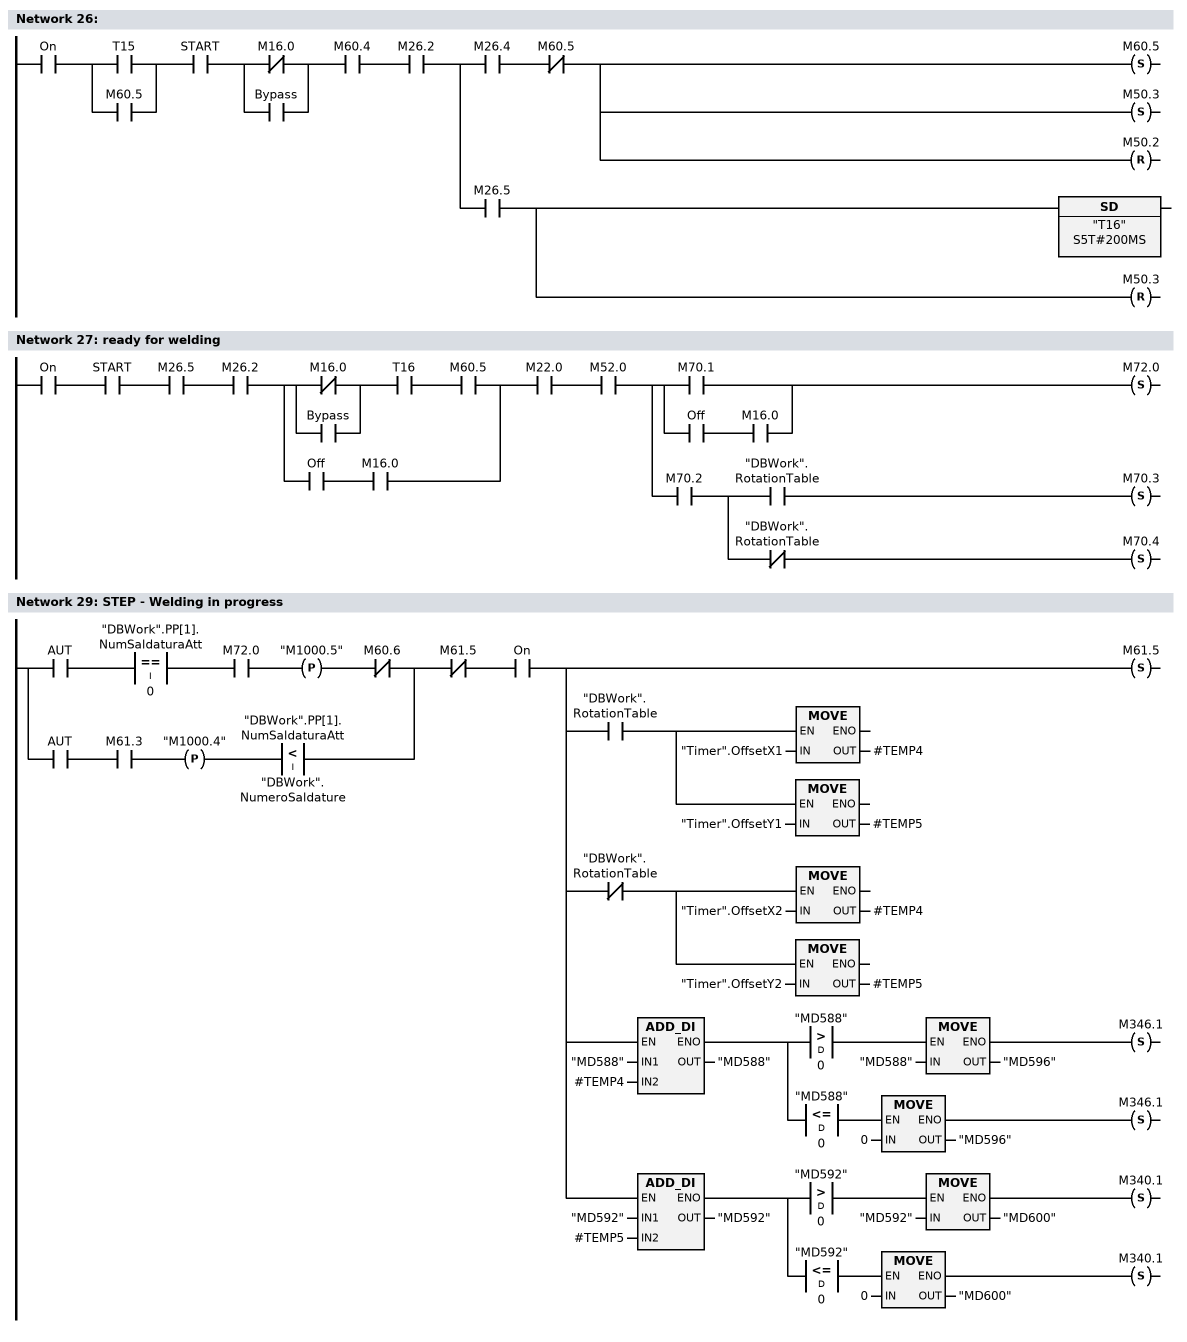
[picture p24: FC14 - AUTOMATIC networks 26-29]
NETWORK
TITLE =
      A     "On";
      A(;
      O     "T15";
      O     "M60.5";
      );
      A     "START";
      A(;
      ON    "M16.0";
      O     "Bypass";
      );
      A     "M60.4";
      A     "M26.2";
      =     L 24.0;
      A     L 24.0;
      A     "M26.4";
      AN    "M60.5";
      S     "M60.5";
      S     "M50.3";
      R     "M50.2";
      A     L 24.0;
      A     "M26.5";
      L     S5T#200MS;
      SD    "T16";
      R     "M50.3";
NETWORK
TITLE = ready for welding
      A     "On";
      A     "START";
      A     "M26.5";
      A     "M26.2";
      A(;
      A(;
      ON    "M16.0";
      O     "Bypass";
      );
      A     "T16";
      A     "M60.5";
      O;
      A     "Off";
      A     "M16.0";
      );
      A     "M22.0";
      A     "M52.0";
      =     L 24.0;
      A     L 24.0;
      A(;
      O     "M70.1";
      O;
      A     "Off";
      A     "M16.0";
      );
      S     "M72.0";
      A     L 24.0;
      A     "M70.2";
      =     L 24.1;
      A     L 24.1;
      A     "DBWork".RotationTable;
      S     "M70.3";
      A     L 24.1;
      AN    "DBWork".RotationTable;
      S     "M70.4";
NETWORK
TITLE =
NETWORK
TITLE = STEP - Welding in progress
      A(;
      A     "AUT";
      A(;
      L     "DBWork".PP[1].NumSaldaturaAtt;
      L     0;
      ==I;
      );
      A     "M72.0";
      FP    "M1000.5";
      AN    "M60.6";
      O(;
      A     "AUT";
      A     "M61.3";
      FP    "M1000.4";
      A(;
      L     "DBWork".PP[1].NumSaldaturaAtt;
      L     "DBWork".NumeroSaldature;
      <I;
      );
      );
      );
      AN    "M61.5";
      A     "On";
      =     L 24.0;
      A     L 24.0;
      BLD   102;
      S     "M61.5";
      A     L 24.0;
      A     "DBWork".RotationTable;
      =     L 24.1;
      A     L 24.1;
      JNB   _00a;
      L     "Timer".OffsetX1;
      T     #TEMP4;
_00a: NOP   0;
      A     L 24.1;
      JNB   _00b;
      L     "Timer".OffsetY1;
      T     #TEMP5;
_00b: NOP   0;
      A     L 24.0;
      AN    "DBWork".RotationTable;
      =     L 24.1;
      A     L 24.1;
      JNB   _00c;
      L     "Timer".OffsetX2;
      T     #TEMP4;
_00c: NOP   0;
      A     L 24.1;
      JNB   _00d;
      L     "Timer".OffsetY2;
      T     #TEMP5;
_00d: NOP   0;
      A     L 24.0;
      JNB   _00e;
      L     "MD588";
      L     #TEMP4;
      +D;
      T     "MD588";
      AN    OV;
      SAVE;
      CLR;
_00e: A     BR;
      =     L 24.1;
      A     L 24.1;
      A(;
      L     "MD588";
      L     0;
      >D;
      );
      JNB   _00f;
      L     "MD588";
      T     "MD596";
      SET;
      SAVE;
      CLR;
_00f: A     BR;
      S     "M346.1";
      A     L 24.1;
      A(;
      L     "MD588";
      L     0;
      <=D;
      );
      JNB   _010;
      L     0;
      T     "MD596";
      SET;
      SAVE;
      CLR;
_010: A     BR;
      S     "M346.1";
      A     L 24.0;
      JNB   _011;
      L     "MD592";
      L     #TEMP5;
      +D;
      T     "MD592";
      AN    OV;
      SAVE;
      CLR;
_011: A     BR;
      =     L 24.1;
      A     L 24.1;
      A(;
      L     "MD592";
      L     0;
      >D;
      );
      JNB   _012;
      L     "MD592";
      T     "MD600";
      SET;
      SAVE;
      CLR;
_012: A     BR;
      S     "M340.1";
      A     L 24.1;
      A(;
      L     "MD592";
      L     0;
      <=D;
      );
      JNB   _013;
      L     0;
      T     "MD600";
      SET;
      SAVE;
      CLR;
_013: A     BR;
      S     "M340.1";
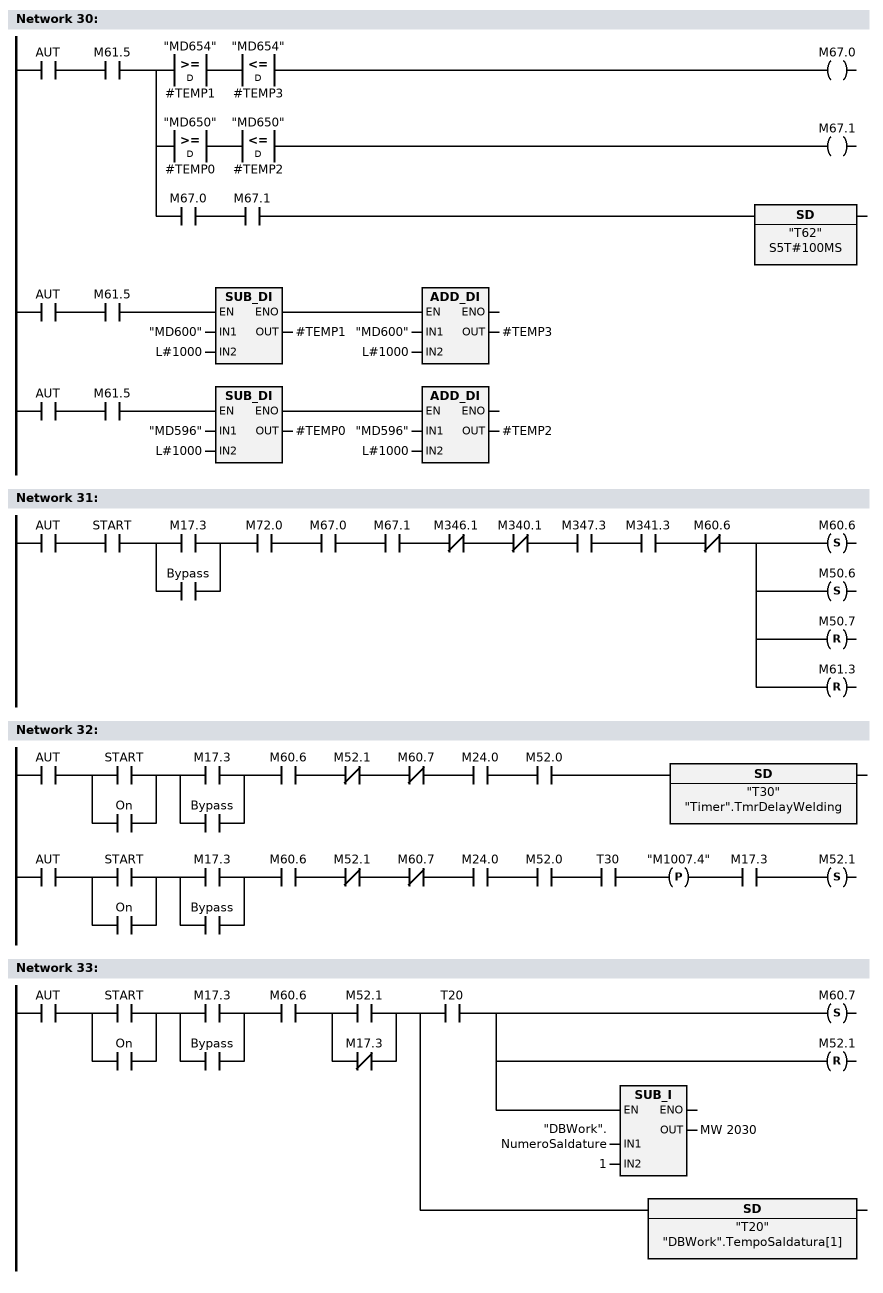
NETWORK
TITLE =
      A     "AUT";
      A     "M61.5";
      =     L 24.0;
      A(;
      A     L 24.0;
      JNB   _014;
      L     "MD600";
      L     L#1000;
      -D;
      T     #TEMP1;
      AN    OV;
      SAVE;
      CLR;
_014: A     BR;
      );
      JNB   _015;
      L     "MD600";
      L     L#1000;
      +D;
      T     #TEMP3;
_015: NOP   0;
      A(;
      A     L 24.0;
      JNB   _016;
      L     "MD596";
      L     L#1000;
      -D;
      T     #TEMP0;
      AN    OV;
      SAVE;
      CLR;
_016: A     BR;
      );
      JNB   _017;
      L     "MD596";
      L     L#1000;
      +D;
      T     #TEMP2;
_017: NOP   0;
      A     L 24.0;
      A(;
      L     "MD654";
      L     #TEMP1;
      >=D;
      );
      A(;
      L     "MD654";
      L     #TEMP3;
      <=D;
      );
      =     "M67.0";
      A     L 24.0;
      A(;
      L     "MD650";
      L     #TEMP0;
      >=D;
      );
      A(;
      L     "MD650";
      L     #TEMP2;
      <=D;
      );
      =     "M67.1";
      A     L 24.0;
      A     "M67.0";
      A     "M67.1";
      L     S5T#100MS;
      SD    "T62";
NETWORK
TITLE =
      A     "AUT";
      A     "START";
      A(;
      O     "M17.3";
      O     "Bypass";
      );
      A     "M72.0";
      A     "M67.0";
      A     "M67.1";
      AN    "M346.1";
      AN    "M340.1";
      A     "M347.3";
      A     "M341.3";
      AN    "M60.6";
      S     "M60.6";
      S     "M50.6";
      R     "M50.7";
      R     "M61.3";
NETWORK
TITLE =
      A     "AUT";
      A(;
      O     "START";
      O     "On";
      );
      A(;
      O     "M17.3";
      O     "Bypass";
      );
      A     "M60.6";
      AN    "M52.1";
      AN    "M60.7";
      A     "M24.0";
      A     "M52.0";
      =     L 24.0;
      A     L 24.0;
      BLD   102;
      L     "Timer".TmrDelayWelding;
      SD    "T30";
      A(;
      A     L 24.0;
      A     "T30";
      FP    "M1007.4";
      );
      A     "M17.3";
      S     "M52.1";
NETWORK
TITLE =
      A     "AUT";
      A(;
      O     "START";
      O     "On";
      );
      A(;
      O     "M17.3";
      O     "Bypass";
      );
      A     "M60.6";
      A(;
      O     "M52.1";
      ON    "M17.3";
      );
      =     L 24.0;
      A     L 24.0;
      A     "T20";
      =     L 24.1;
      A     L 24.1;
      BLD   102;
      S     "M60.7";
      A     L 24.1;
      BLD   102;
      R     "M52.1";
      A     L 24.1;
      JNB   _018;
      L     "DBWork".NumeroSaldature;
      L     1;
      -I;
      T     MW 2030;
_018: NOP   0;
      A     L 24.0;
      BLD   102;
      L     "DBWork".TempoSaldatura[1];
      SD    "T20";
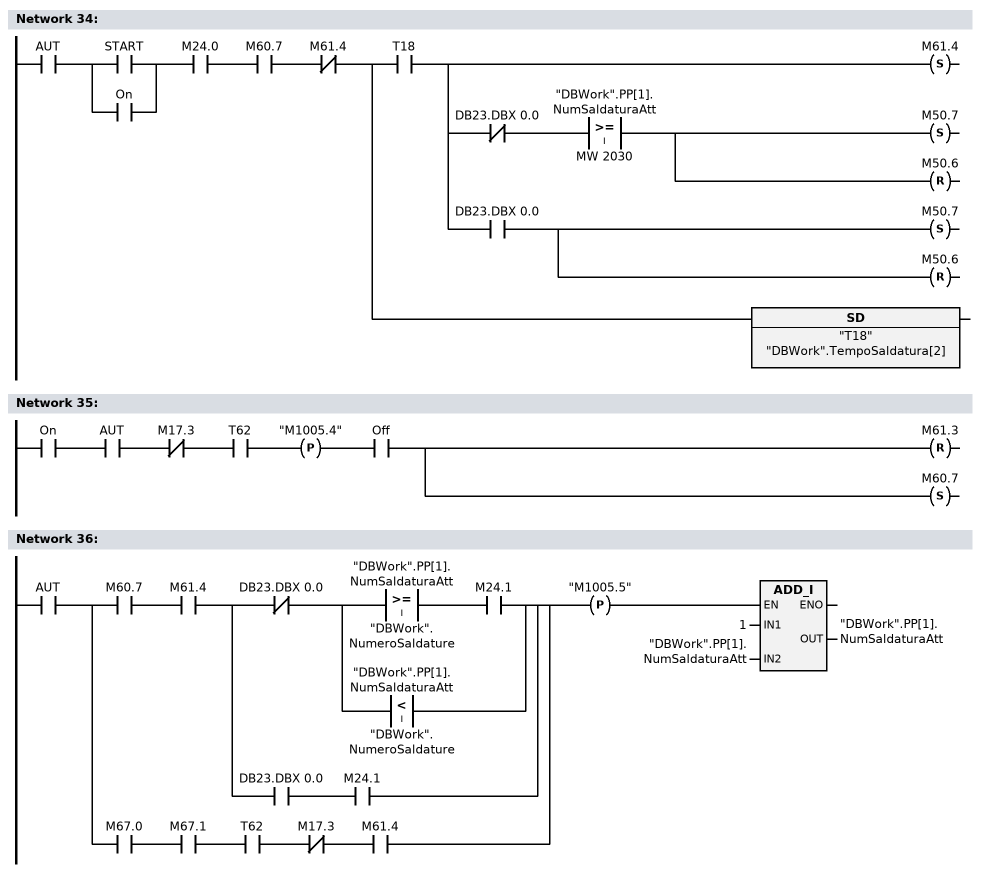
NETWORK
TITLE =
      A     "AUT";
      A(;
      O     "START";
      O     "On";
      );
      A     "M24.0";
      A     "M60.7";
      AN    "M61.4";
      =     L 24.0;
      A     L 24.0;
      A     "T18";
      =     L 24.1;
      A     L 24.1;
      BLD   102;
      S     "M61.4";
      A     L 24.1;
      AN    DB23.DBX 0.0;
      A(;
      L     "DBWork".PP[1].NumSaldaturaAtt;
      L     MW 2030;
      >=I;
      );
      S     "M50.7";
      R     "M50.6";
      A     L 24.1;
      A     DB23.DBX 0.0;
      S     "M50.7";
      R     "M50.6";
      A     L 24.0;
      BLD   102;
      L     "DBWork".TempoSaldatura[2];
      SD    "T18";
NETWORK
TITLE =
      A     "On";
      A     "AUT";
      AN    "M17.3";
      A     "T62";
      FP    "M1005.4";
      A     "Off";
      R     "M61.3";
      S     "M60.7";
NETWORK
TITLE =
      A     "AUT";
      A(;
      A     "M60.7";
      A     "M61.4";
      A(;
      AN    DB23.DBX 0.0;
      A(;
      A(;
      L     "DBWork".PP[1].NumSaldaturaAtt;
      L     "DBWork".NumeroSaldature;
      >=I;
      );
      A     "M24.1";
      O(;
      L     "DBWork".PP[1].NumSaldaturaAtt;
      L     "DBWork".NumeroSaldature;
      <I;
      );
      );
      O;
      A     DB23.DBX 0.0;
      A     "M24.1";
      );
      O;
      A     "M67.0";
      A     "M67.1";
      A     "T62";
      AN    "M17.3";
      A     "M61.4";
      );
      FP    "M1005.5";
      JNB   _019;
      L     1;
      L     "DBWork".PP[1].NumSaldaturaAtt;
      +I;
      T     "DBWork".PP[1].NumSaldaturaAtt;
_019: NOP   0;
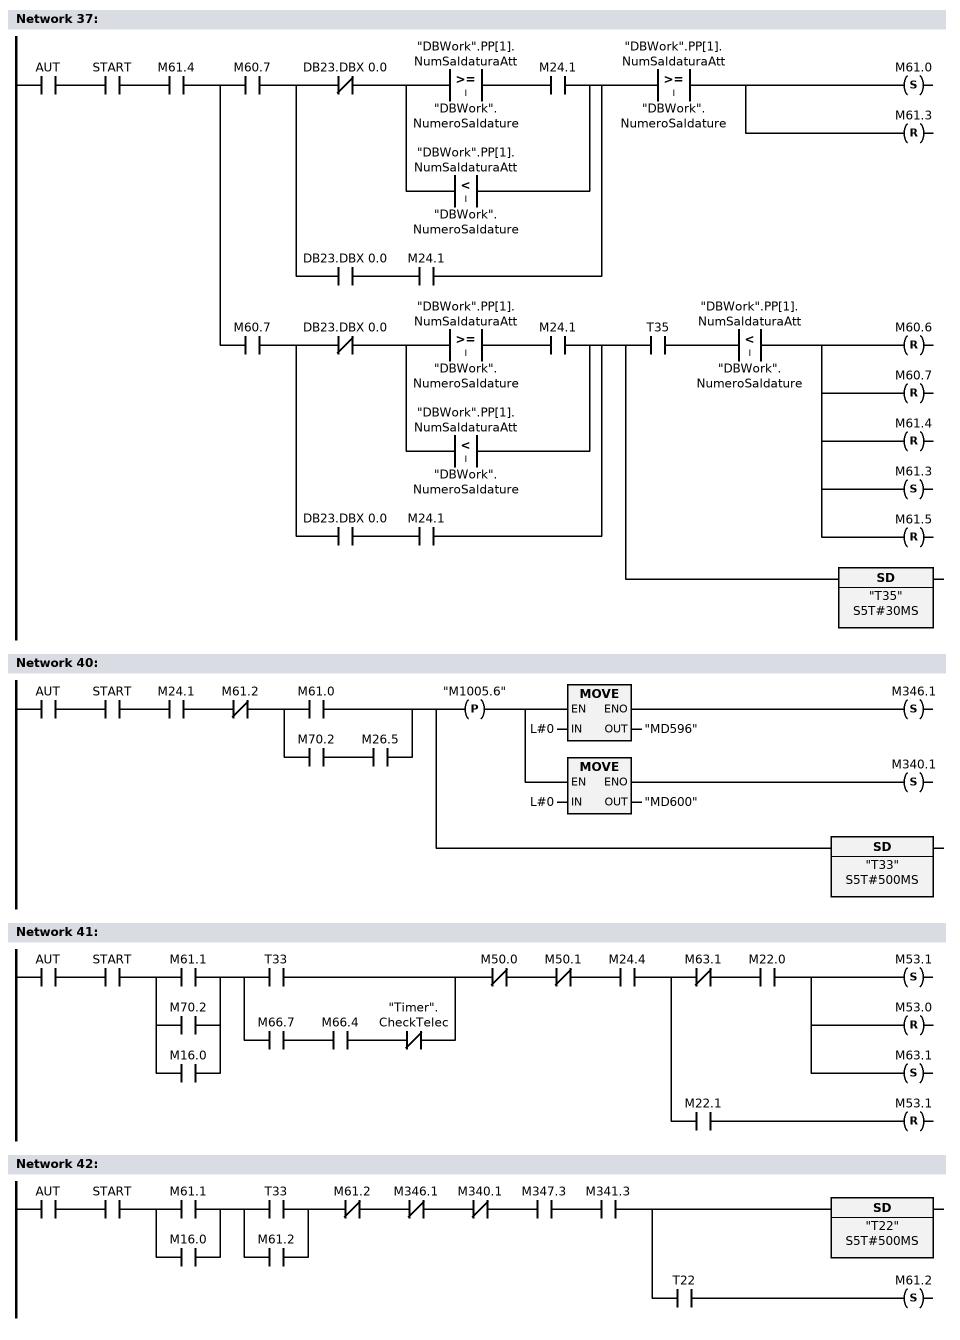
NETWORK
TITLE =
      A     "AUT";
      A     "START";
      A     "M61.4";
      =     L 24.0;
      A     L 24.0;
      A     "M60.7";
      A(;
      AN    DB23.DBX 0.0;
      A(;
      A(;
      L     "DBWork".PP[1].NumSaldaturaAtt;
      L     "DBWork".NumeroSaldature;
      >=I;
      );
      A     "M24.1";
      O(;
      L     "DBWork".PP[1].NumSaldaturaAtt;
      L     "DBWork".NumeroSaldature;
      <I;
      );
      );
      O;
      A     DB23.DBX 0.0;
      A     "M24.1";
      );
      A(;
      L     "DBWork".PP[1].NumSaldaturaAtt;
      L     "DBWork".NumeroSaldature;
      >=I;
      );
      S     "M61.0";
      R     "M61.3";
      A     L 24.0;
      A     "M60.7";
      A(;
      AN    DB23.DBX 0.0;
      A(;
      A(;
      L     "DBWork".PP[1].NumSaldaturaAtt;
      L     "DBWork".NumeroSaldature;
      >=I;
      );
      A     "M24.1";
      O(;
      L     "DBWork".PP[1].NumSaldaturaAtt;
      L     "DBWork".NumeroSaldature;
      <I;
      );
      );
      O;
      A     DB23.DBX 0.0;
      A     "M24.1";
      );
      =     L 24.1;
      A     L 24.1;
      A     "T35";
      A(;
      L     "DBWork".PP[1].NumSaldaturaAtt;
      L     "DBWork".NumeroSaldature;
      <I;
      );
      R     "M60.6";
      R     "M60.7";
      R     "M61.4";
      S     "M61.3";
      R     "M61.5";
      A     L 24.1;
      BLD   102;
      L     S5T#30MS;
      SD    "T35";
NETWORK
TITLE =
NETWORK
TITLE =
NETWORK
TITLE =
      A     "AUT";
      A     "START";
      A     "M24.1";
      AN    "M61.2";
      A(;
      O     "M61.0";
      O;
      A     "M70.2";
      A     "M26.5";
      );
      =     L 24.0;
      A     L 24.0;
      FP    "M1005.6";
      =     L 24.1;
      A     L 24.1;
      JNB   _01a;
      L     L#0;
      T     "MD596";
      SET;
      SAVE;
      CLR;
_01a: A     BR;
      S     "M346.1";
      A     L 24.1;
      JNB   _01b;
      L     L#0;
      T     "MD600";
      SET;
      SAVE;
      CLR;
_01b: A     BR;
      S     "M340.1";
      A     L 24.0;
      BLD   102;
      L     S5T#500MS;
      SD    "T33";
NETWORK
TITLE =
      A     "AUT";
      A     "START";
      A(;
      O     "M61.1";
      O     "M70.2";
      O     "M16.0";
      );
      A(;
      O     "T33";
      O;
      A     "M66.7";
      A     "M66.4";
      AN    "Timer".CheckTelec;
      );
      AN    "M50.0";
      AN    "M50.1";
      A     "M24.4";
      =     L 24.0;
      A     L 24.0;
      AN    "M63.1";
      A     "M22.0";
      S     "M53.1";
      R     "M53.0";
      S     "M63.1";
      A     L 24.0;
      A     "M22.1";
      R     "M53.1";
NETWORK
TITLE =
      A     "AUT";
      A     "START";
      A(;
      O     "M61.1";
      O     "M16.0";
      );
      A(;
      O     "T33";
      O     "M61.2";
      );
      AN    "M61.2";
      AN    "M346.1";
      AN    "M340.1";
      A     "M347.3";
      A     "M341.3";
      =     L 24.0;
      A     L 24.0;
      BLD   102;
      L     S5T#500MS;
      SD    "T22";
      A     L 24.0;
      A     "T22";
      S     "M61.2";
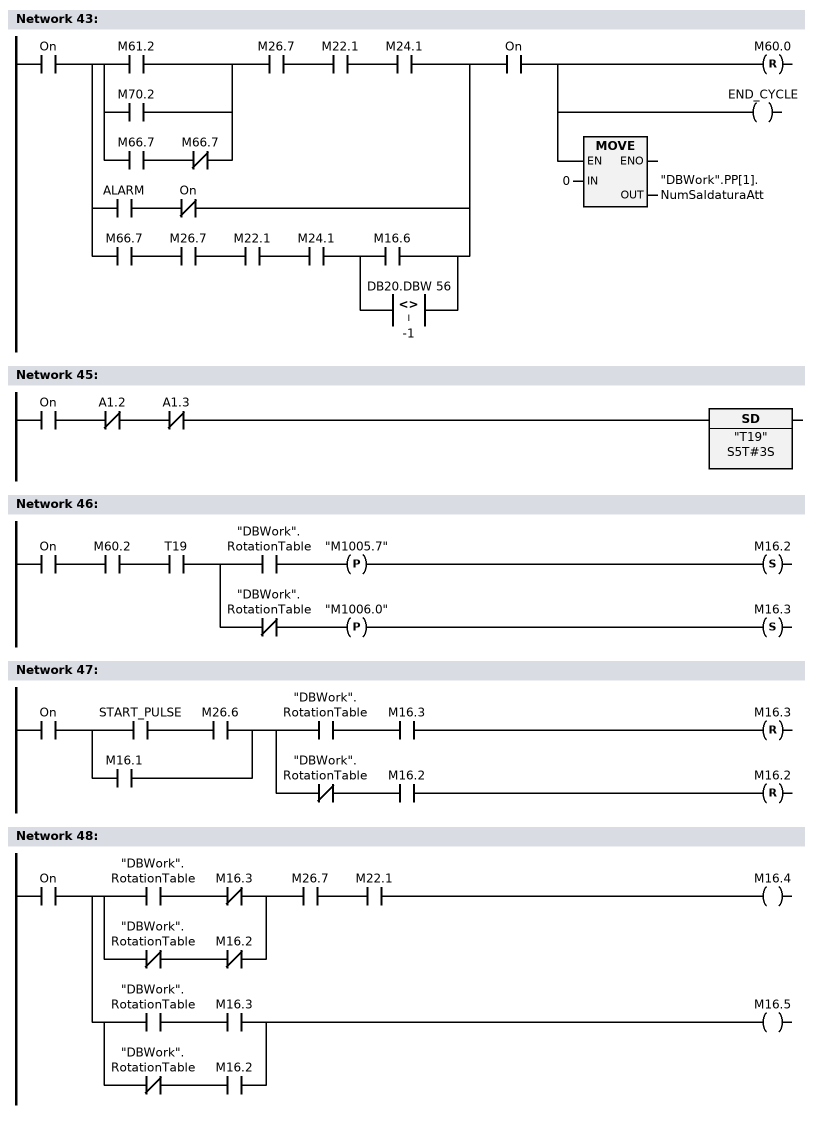
NETWORK
TITLE =
      A     "On";
      A(;
      A(;
      O     "M61.2";
      O     "M70.2";
      O;
      A     "M66.7";
      AN    "M66.7";
      );
      A     "M26.7";
      A     "M22.1";
      A     "M24.1";
      O;
      A     "ALARM";
      AN    "On";
      O;
      A     "M66.7";
      A     "M26.7";
      A     "M22.1";
      A     "M24.1";
      A(;
      O     "M16.6";
      O(;
      L     DB20.DBW 56;
      L     -1;
      <>I;
      );
      );
      );
      A     "On";
      =     L 24.0;
      A     L 24.0;
      BLD   102;
      R     "M60.0";
      A     L 24.0;
      BLD   102;
      =     "END_CYCLE";
      A     L 24.0;
      JNB   _01c;
      L     0;
      T     "DBWork".PP[1].NumSaldaturaAtt;
_01c: NOP   0;
NETWORK
TITLE =
NETWORK
TITLE =
      A     "On";
      AN    "A1.2";
      AN    "A1.3";
      L     S5T#3S;
      SD    "T19";
NETWORK
TITLE =
      A     "On";
      A     "M60.2";
      A     "T19";
      =     L 24.0;
      A     L 24.0;
      A     "DBWork".RotationTable;
      FP    "M1005.7";
      S     "M16.2";
      A     L 24.0;
      AN    "DBWork".RotationTable;
      FP    "M1006.0";
      S     "M16.3";
NETWORK
TITLE =
      A     "On";
      A(;
      A     "START_PULSE";
      A     "M26.6";
      O     "M16.1";
      );
      =     L 24.0;
      A     L 24.0;
      A     "DBWork".RotationTable;
      A     "M16.3";
      R     "M16.3";
      A     L 24.0;
      AN    "DBWork".RotationTable;
      A     "M16.2";
      R     "M16.2";
NETWORK
TITLE =
      A     "On";
      =     L 24.0;
      A     L 24.0;
      A(;
      A     "DBWork".RotationTable;
      AN    "M16.3";
      O;
      AN    "DBWork".RotationTable;
      AN    "M16.2";
      );
      A     "M26.7";
      A     "M22.1";
      =     "M16.4";
      A     L 24.0;
      A(;
      A     "DBWork".RotationTable;
      A     "M16.3";
      O;
      AN    "DBWork".RotationTable;
      A     "M16.2";
      );
      =     "M16.5";
END_FUNCTION

FUNCTION "FC16 - ALARMS" : VOID	// FC 16
VERSION : 0.1
VAR_TEMP
  TEMP0 : BOOL ;
END_VAR
BEGIN
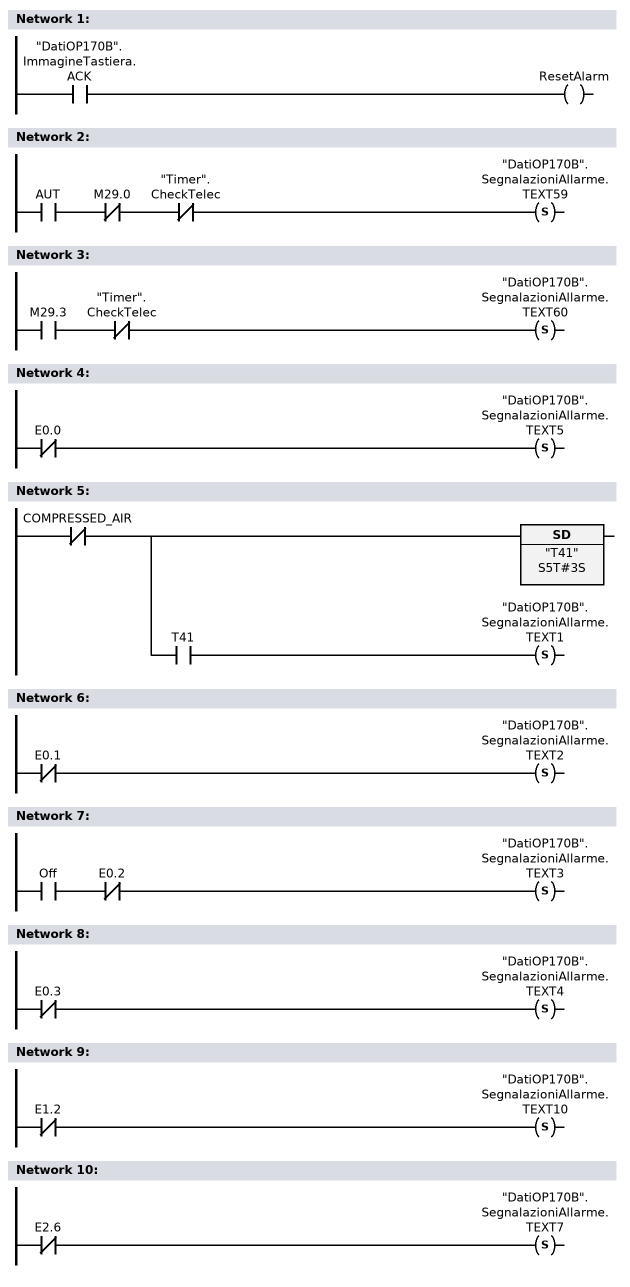
NETWORK
TITLE =
      A     "DatiOP170B".ImmagineTastiera.ACK;
      =     "ResetAlarm";
NETWORK
TITLE =
      A     "AUT";
      AN    "M29.0";
      AN    "Timer".CheckTelec;
      S     "DatiOP170B".SegnalazioniAllarme.TEXT59;
NETWORK
TITLE =
      A     "M29.3";
      AN    "Timer".CheckTelec;
      S     "DatiOP170B".SegnalazioniAllarme.TEXT60;
NETWORK
TITLE =
      AN    "E0.0";
      S     "DatiOP170B".SegnalazioniAllarme.TEXT5;
NETWORK
TITLE =
      AN    "COMPRESSED_AIR";
      =     L 1.0;
      A     L 1.0;
      BLD   102;
      L     S5T#3S;
      SD    "T41";
      A     L 1.0;
      A     "T41";
      S     "DatiOP170B".SegnalazioniAllarme.TEXT1;
NETWORK
TITLE =
      AN    "E0.1";
      S     "DatiOP170B".SegnalazioniAllarme.TEXT2;
NETWORK
TITLE =
      A     "Off";
      AN    "E0.2";
      S     "DatiOP170B".SegnalazioniAllarme.TEXT3;
NETWORK
TITLE =
      AN    "E0.3";
      S     "DatiOP170B".SegnalazioniAllarme.TEXT4;
NETWORK
TITLE =
      AN    "E1.2";
      S     "DatiOP170B".SegnalazioniAllarme.TEXT10;
NETWORK
TITLE =
      AN    "E2.6";
      S     "DatiOP170B".SegnalazioniAllarme.TEXT7;
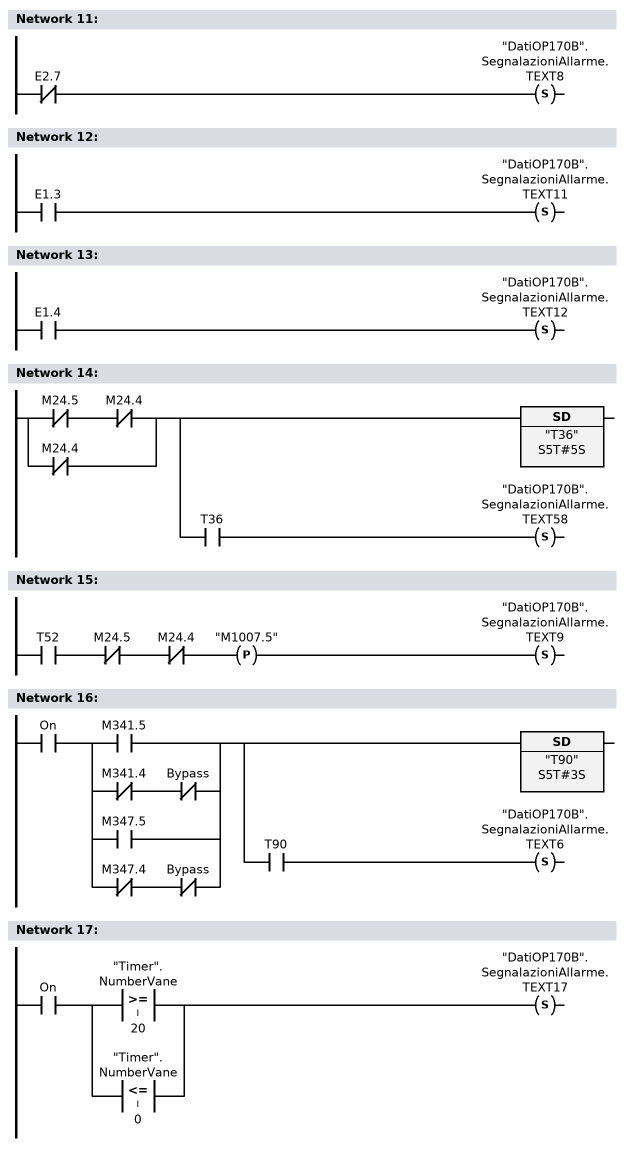
NETWORK
TITLE =
      AN    "E2.7";
      S     "DatiOP170B".SegnalazioniAllarme.TEXT8;
NETWORK
TITLE =
      A     "E1.3";
      S     "DatiOP170B".SegnalazioniAllarme.TEXT11;
NETWORK
TITLE =
      A     "E1.4";
      S     "DatiOP170B".SegnalazioniAllarme.TEXT12;
NETWORK
TITLE =
      AN    "M24.5";
      AN    "M24.4";
      ON    "M24.4";
      =     L 1.0;
      A     L 1.0;
      BLD   102;
      L     S5T#5S;
      SD    "T36";
      A     L 1.0;
      A     "T36";
      S     "DatiOP170B".SegnalazioniAllarme.TEXT58;
NETWORK
TITLE =
      A     "T52";
      AN    "M24.5";
      AN    "M24.4";
      FP    "M1007.5";
      S     "DatiOP170B".SegnalazioniAllarme.TEXT9;
NETWORK
TITLE =
      A     "On";
      A(;
      O     "M341.5";
      O;
      AN    "M341.4";
      AN    "Bypass";
      O     "M347.5";
      O;
      AN    "M347.4";
      AN    "Bypass";
      );
      =     L 1.0;
      A     L 1.0;
      BLD   102;
      L     S5T#3S;
      SD    "T90";
      A     L 1.0;
      A     "T90";
      S     "DatiOP170B".SegnalazioniAllarme.TEXT6;
NETWORK
TITLE =
      A     "On";
      A(;
      O(;
      L     "Timer".NumberVane;
      L     20;
      >=I;
      );
      O(;
      L     "Timer".NumberVane;
      L     0;
      <=I;
      );
      );
      S     "DatiOP170B".SegnalazioniAllarme.TEXT17;
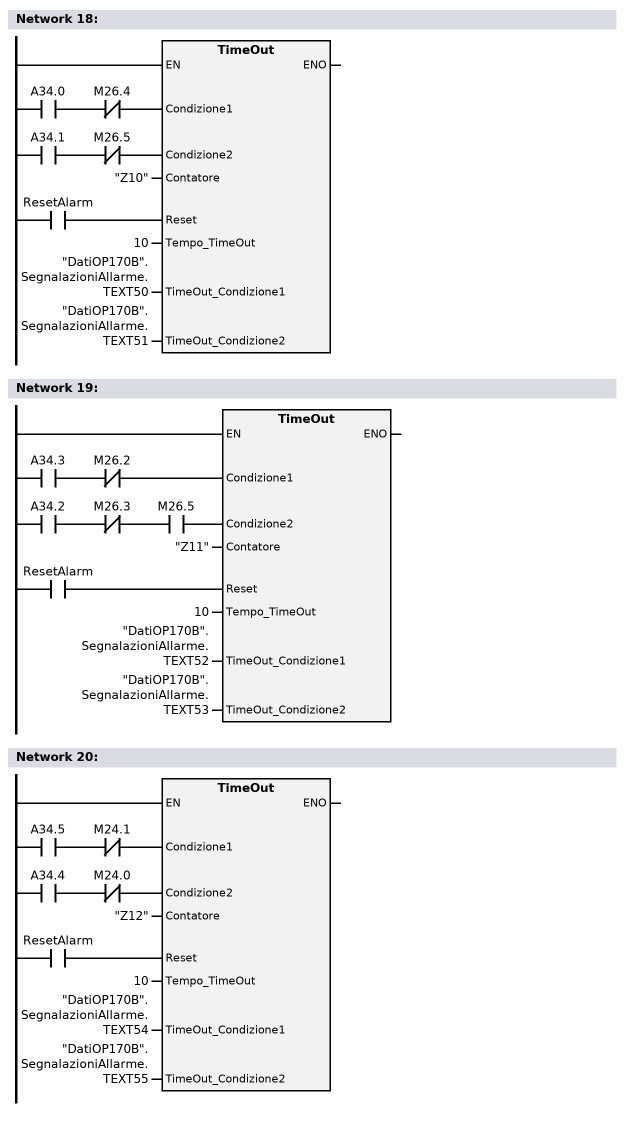
NETWORK
TITLE =
      A     "A34.0";
      AN    "M26.4";
      =     L 1.0;
      BLD   103;
      A     "A34.1";
      AN    "M26.5";
      =     L 1.1;
      BLD   103;
      A     "ResetAlarm";
      =     L 1.2;
      BLD   103;
      CALL  "TimeOut" (
           Condizione1              := L 1.0,
           Condizione2              := L 1.1,
           Contatore                := "Z10",
           Reset                    := L 1.2,
           Tempo_TimeOut            := 10,
           TimeOut_Condizione1      := "DatiOP170B".SegnalazioniAllarme.TEXT50,
           TimeOut_Condizione2      := "DatiOP170B".SegnalazioniAllarme.TEXT51);
      NOP   0;
NETWORK
TITLE =
      A     "A34.3";
      AN    "M26.2";
      =     L 1.0;
      BLD   103;
      A     "A34.2";
      AN    "M26.3";
      A     "M26.5";
      =     L 1.1;
      BLD   103;
      A     "ResetAlarm";
      =     L 1.2;
      BLD   103;
      CALL  "TimeOut" (
           Condizione1              := L 1.0,
           Condizione2              := L 1.1,
           Contatore                := "Z11",
           Reset                    := L 1.2,
           Tempo_TimeOut            := 10,
           TimeOut_Condizione1      := "DatiOP170B".SegnalazioniAllarme.TEXT52,
           TimeOut_Condizione2      := "DatiOP170B".SegnalazioniAllarme.TEXT53);
      NOP   0;
NETWORK
TITLE =
      A     "A34.5";
      AN    "M24.1";
      =     L 1.0;
      BLD   103;
      A     "A34.4";
      AN    "M24.0";
      =     L 1.1;
      BLD   103;
      A     "ResetAlarm";
      =     L 1.2;
      BLD   103;
      CALL  "TimeOut" (
           Condizione1              := L 1.0,
           Condizione2              := L 1.1,
           Contatore                := "Z12",
           Reset                    := L 1.2,
           Tempo_TimeOut            := 10,
           TimeOut_Condizione1      := "DatiOP170B".SegnalazioniAllarme.TEXT54,
           TimeOut_Condizione2      := "DatiOP170B".SegnalazioniAllarme.TEXT55);
      NOP   0;
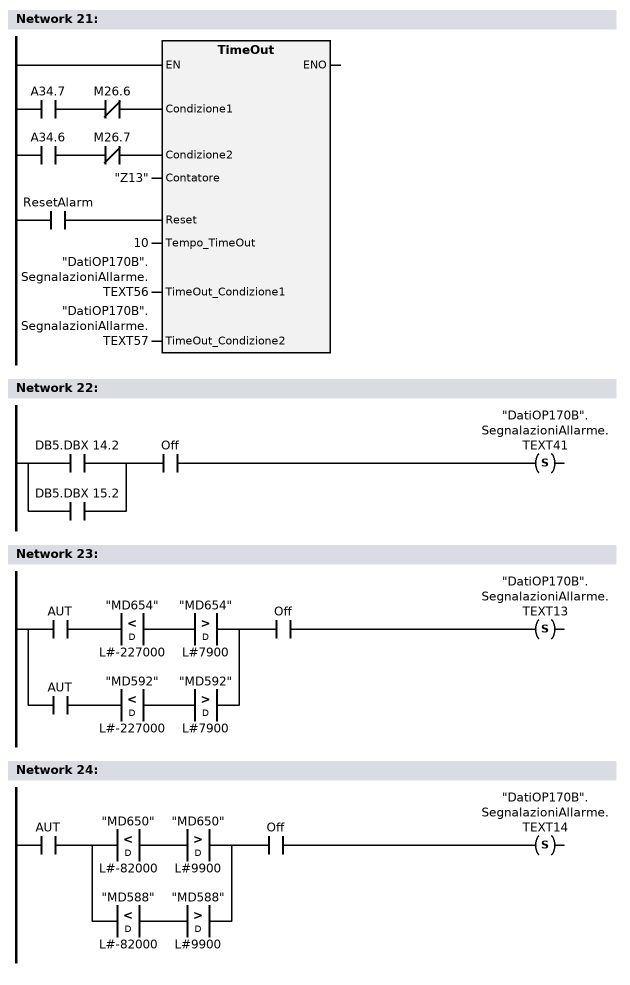
NETWORK
TITLE =
      A     "A34.7";
      AN    "M26.6";
      =     L 1.0;
      BLD   103;
      A     "A34.6";
      AN    "M26.7";
      =     L 1.1;
      BLD   103;
      A     "ResetAlarm";
      =     L 1.2;
      BLD   103;
      CALL  "TimeOut" (
           Condizione1              := L 1.0,
           Condizione2              := L 1.1,
           Contatore                := "Z13",
           Reset                    := L 1.2,
           Tempo_TimeOut            := 10,
           TimeOut_Condizione1      := "DatiOP170B".SegnalazioniAllarme.TEXT56,
           TimeOut_Condizione2      := "DatiOP170B".SegnalazioniAllarme.TEXT57);
      NOP   0;
NETWORK
TITLE =
      A(;
      O     DB5.DBX 14.2;
      O     DB5.DBX 15.2;
      );
      A     "Off";
      S     "DatiOP170B".SegnalazioniAllarme.TEXT41;
NETWORK
TITLE =
      A(;
      A     "AUT";
      A(;
      L     "MD654";
      L     L#-227000;
      <D;
      );
      A(;
      L     "MD654";
      L     L#7900;
      >D;
      );
      O;
      A     "AUT";
      A(;
      L     "MD592";
      L     L#-227000;
      <D;
      );
      A(;
      L     "MD592";
      L     L#7900;
      >D;
      );
      );
      A     "Off";
      S     "DatiOP170B".SegnalazioniAllarme.TEXT13;
NETWORK
TITLE =
      A     "AUT";
      A(;
      A(;
      L     "MD650";
      L     L#-82000;
      <D;
      );
      A(;
      L     "MD650";
      L     L#9900;
      >D;
      );
      O;
      A(;
      L     "MD588";
      L     L#-82000;
      <D;
      );
      A(;
      L     "MD588";
      L     L#9900;
      >D;
      );
      );
      A     "Off";
      S     "DatiOP170B".SegnalazioniAllarme.TEXT14;
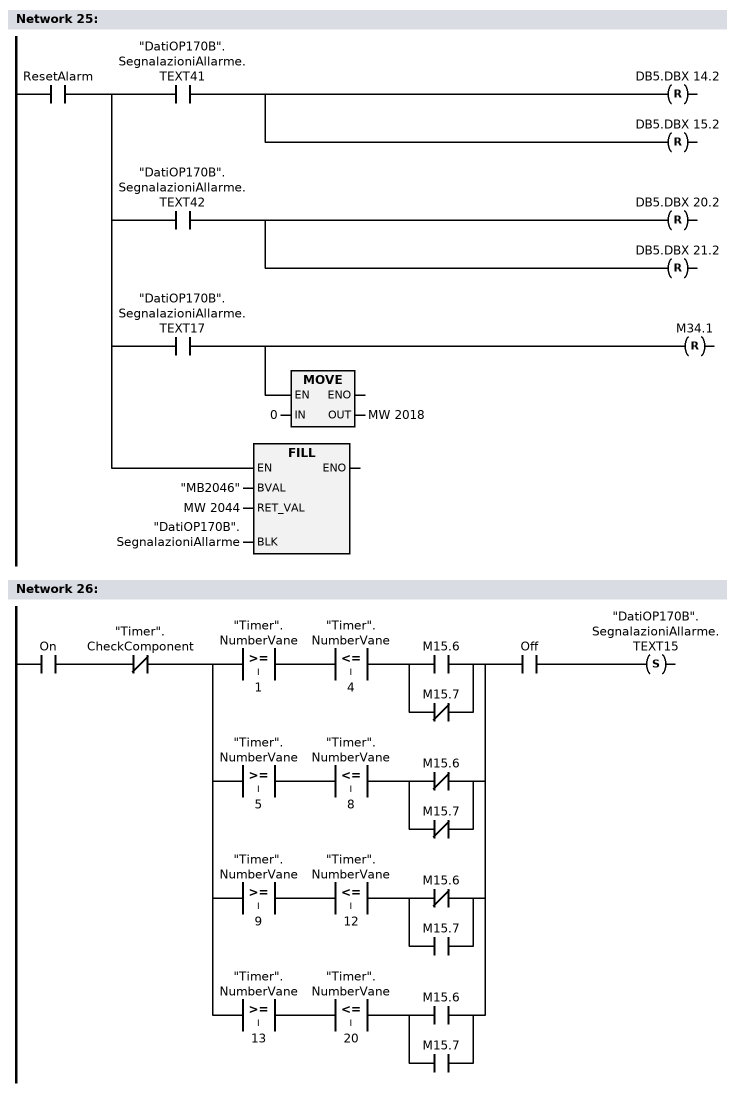
NETWORK
TITLE =
      A     "ResetAlarm";
      =     L 1.0;
      A     L 1.0;
      A     "DatiOP170B".SegnalazioniAllarme.TEXT41;
      R     DB5.DBX 14.2;
      R     DB5.DBX 15.2;
      A     L 1.0;
      A     "DatiOP170B".SegnalazioniAllarme.TEXT42;
      R     DB5.DBX 20.2;
      R     DB5.DBX 21.2;
      A     L 1.0;
      A     "DatiOP170B".SegnalazioniAllarme.TEXT17;
      =     L 1.1;
      A     L 1.1;
      BLD   102;
      R     "M34.1";
      A     L 1.1;
      JNB   _001;
      L     0;
      T     MW 2018;
_001: NOP   0;
      A     L 1.0;
      JNB   _002;
      CALL  "FILL" (
           BVAL                     := "MB2046",
           RET_VAL                  := MW 2044,
           BLK                      := "DatiOP170B".SegnalazioniAllarme);
_002: NOP   0;
NETWORK
TITLE =
      A     "On";
      AN    "Timer".CheckComponent;
      A(;
      A(;
      L     "Timer".NumberVane;
      L     1;
      >=I;
      );
      A(;
      L     "Timer".NumberVane;
      L     4;
      <=I;
      );
      A(;
      O     "M15.6";
      ON    "M15.7";
      );
      O;
      A(;
      L     "Timer".NumberVane;
      L     5;
      >=I;
      );
      A(;
      L     "Timer".NumberVane;
      L     8;
      <=I;
      );
      A(;
      ON    "M15.6";
      ON    "M15.7";
      );
      O;
      A(;
      L     "Timer".NumberVane;
      L     9;
      >=I;
      );
      A(;
      L     "Timer".NumberVane;
      L     12;
      <=I;
      );
      A(;
      ON    "M15.6";
      O     "M15.7";
      );
      O;
      A(;
      L     "Timer".NumberVane;
      L     13;
      >=I;
      );
      A(;
      L     "Timer".NumberVane;
      L     20;
      <=I;
      );
      A(;
      O     "M15.6";
      O     "M15.7";
      );
      );
      A     "Off";
      S     "DatiOP170B".SegnalazioniAllarme.TEXT15;
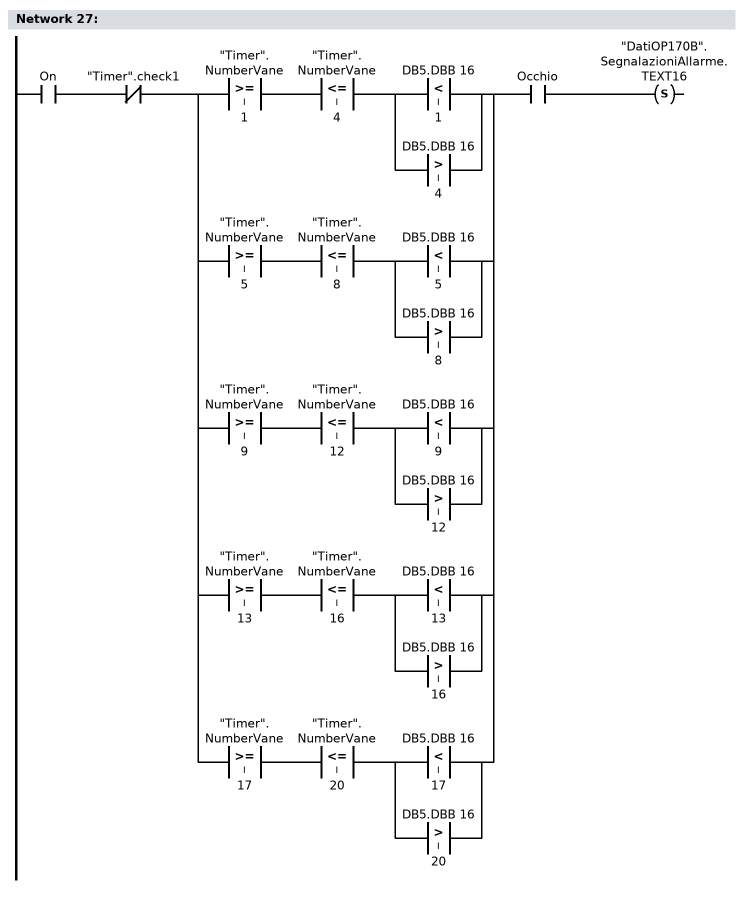
NETWORK
TITLE =
      A     "On";
      AN    "Timer".check1;
      A(;
      A(;
      L     "Timer".NumberVane;
      L     1;
      >=I;
      );
      A(;
      L     "Timer".NumberVane;
      L     4;
      <=I;
      );
      A(;
      O(;
      L     DB5.DBB 16;
      L     1;
      <I;
      );
      O(;
      L     DB5.DBB 16;
      L     4;
      >I;
      );
      );
      O;
      A(;
      L     "Timer".NumberVane;
      L     5;
      >=I;
      );
      A(;
      L     "Timer".NumberVane;
      L     8;
      <=I;
      );
      A(;
      O(;
      L     DB5.DBB 16;
      L     5;
      <I;
      );
      O(;
      L     DB5.DBB 16;
      L     8;
      >I;
      );
      );
      O;
      A(;
      L     "Timer".NumberVane;
      L     9;
      >=I;
      );
      A(;
      L     "Timer".NumberVane;
      L     12;
      <=I;
      );
      A(;
      O(;
      L     DB5.DBB 16;
      L     9;
      <I;
      );
      O(;
      L     DB5.DBB 16;
      L     12;
      >I;
      );
      );
      O;
      A(;
      L     "Timer".NumberVane;
      L     13;
      >=I;
      );
      A(;
      L     "Timer".NumberVane;
      L     16;
      <=I;
      );
      A(;
      O(;
      L     DB5.DBB 16;
      L     13;
      <I;
      );
      O(;
      L     DB5.DBB 16;
      L     16;
      >I;
      );
      );
      O;
      A(;
      L     "Timer".NumberVane;
      L     17;
      >=I;
      );
      A(;
      L     "Timer".NumberVane;
      L     20;
      <=I;
      );
      A(;
      O(;
      L     DB5.DBB 16;
      L     17;
      <I;
      );
      O(;
      L     DB5.DBB 16;
      L     20;
      >I;
      );
      );
      );
      A     "Occhio";
      S     "DatiOP170B".SegnalazioniAllarme.TEXT16;
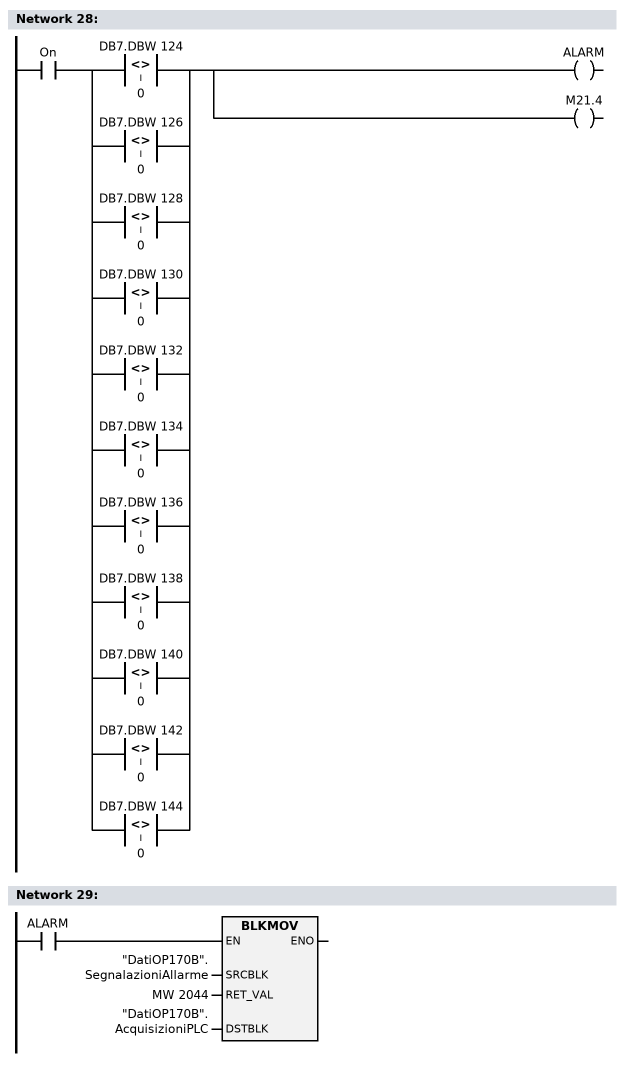
NETWORK
TITLE =
      A     "On";
      A(;
      O(;
      L     DB7.DBW 124;
      L     0;
      <>I;
      );
      O(;
      L     DB7.DBW 126;
      L     0;
      <>I;
      );
      O(;
      L     DB7.DBW 128;
      L     0;
      <>I;
      );
      O(;
      L     DB7.DBW 130;
      L     0;
      <>I;
      );
      O(;
      L     DB7.DBW 132;
      L     0;
      <>I;
      );
      O(;
      L     DB7.DBW 134;
      L     0;
      <>I;
      );
      O(;
      L     DB7.DBW 136;
      L     0;
      <>I;
      );
      O(;
      L     DB7.DBW 138;
      L     0;
      <>I;
      );
      O(;
      L     DB7.DBW 140;
      L     0;
      <>I;
      );
      O(;
      L     DB7.DBW 142;
      L     0;
      <>I;
      );
      O(;
      L     DB7.DBW 144;
      L     0;
      <>I;
      );
      );
      =     "ALARM";
      =     "M21.4";
NETWORK
TITLE =
      A     "ALARM";
      JNB   _003;
      CALL  "BLKMOV" (
           SRCBLK                   := "DatiOP170B".SegnalazioniAllarme,
           RET_VAL                  := MW 2044,
           DSTBLK                   := "DatiOP170B".AcquisizioniPLC);
_003: NOP   0;
END_FUNCTION

FUNCTION "FC17 - OPERATOR PANNEL" : VOID	// FC 17
VERSION : 0.1
BEGIN
// (block stored without names or comments; labels and parameter names are numbered)
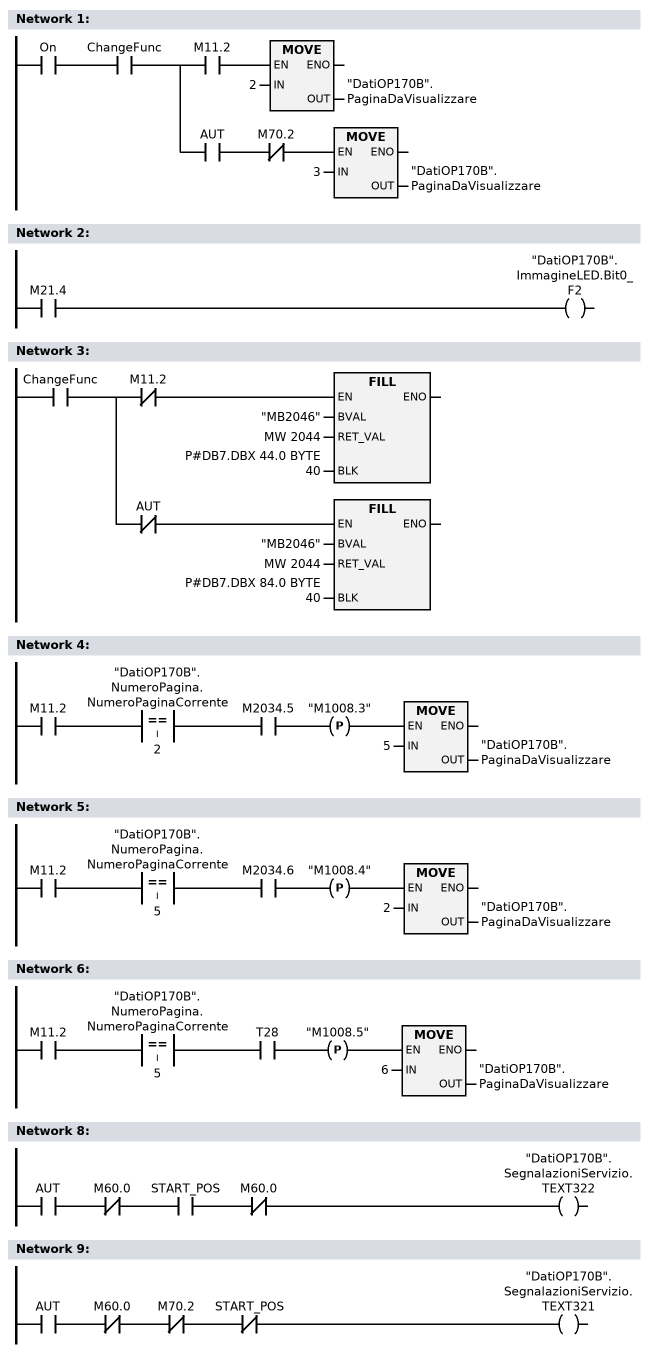
NETWORK
TITLE =
      A     "On";
      A     "ChangeFunc";
      =     L 0.0;
      A     L 0.0;
      A     "M11.2";
      JNB   M001;
      L     2;
      T     "DatiOP170B".PaginaDaVisualizzare;
M001: NOP   0;
      A     L 0.0;
      A     "AUT";
      AN    "M70.2";
      JNB   M002;
      L     3;
      T     "DatiOP170B".PaginaDaVisualizzare;
M002: NOP   0;
NETWORK
TITLE =
      A     "M21.4";
      =     "DatiOP170B".ImmagineLED.Bit0_F2;
NETWORK
TITLE =
      A     "ChangeFunc";
      =     L 0.0;
      A     L 0.0;
      AN    "M11.2";
      JNB   M003;
      CALL  "FILL" (
           BVAL                     := "MB2046",
           RET_VAL                  := MW 2044,
           BLK                      := P#DB7.DBX 44.0 BYTE 40);
M003: NOP   0;
      A     L 0.0;
      AN    "AUT";
      JNB   M004;
      CALL  "FILL" (
           BVAL                     := "MB2046",
           RET_VAL                  := MW 2044,
           BLK                      := P#DB7.DBX 84.0 BYTE 40);
M004: NOP   0;
NETWORK
TITLE =
      A     "M11.2";
      A(;
      L     "DatiOP170B".NumeroPagina.NumeroPaginaCorrente;
      L     2;
      ==I;
      );
      A     "M2034.5";
      FP    "M1008.3";
      JNB   M005;
      L     5;
      T     "DatiOP170B".PaginaDaVisualizzare;
M005: NOP   0;
NETWORK
TITLE =
      A     "M11.2";
      A(;
      L     "DatiOP170B".NumeroPagina.NumeroPaginaCorrente;
      L     5;
      ==I;
      );
      A     "M2034.6";
      FP    "M1008.4";
      JNB   M006;
      L     2;
      T     "DatiOP170B".PaginaDaVisualizzare;
M006: NOP   0;
NETWORK
TITLE =
      A     "M11.2";
      A(;
      L     "DatiOP170B".NumeroPagina.NumeroPaginaCorrente;
      L     5;
      ==I;
      );
      A     "T28";
      FP    "M1008.5";
      JNB   M007;
      L     6;
      T     "DatiOP170B".PaginaDaVisualizzare;
M007: NOP   0;
NETWORK
TITLE =
NETWORK
TITLE =
      A     "AUT";
      AN    "M60.0";
      A     "START_POS";
      AN    "M60.0";
      =     "DatiOP170B".SegnalazioniServizio.TEXT322;
NETWORK
TITLE =
      A     "AUT";
      AN    "M60.0";
      AN    "M70.2";
      AN    "START_POS";
      =     "DatiOP170B".SegnalazioniServizio.TEXT321;
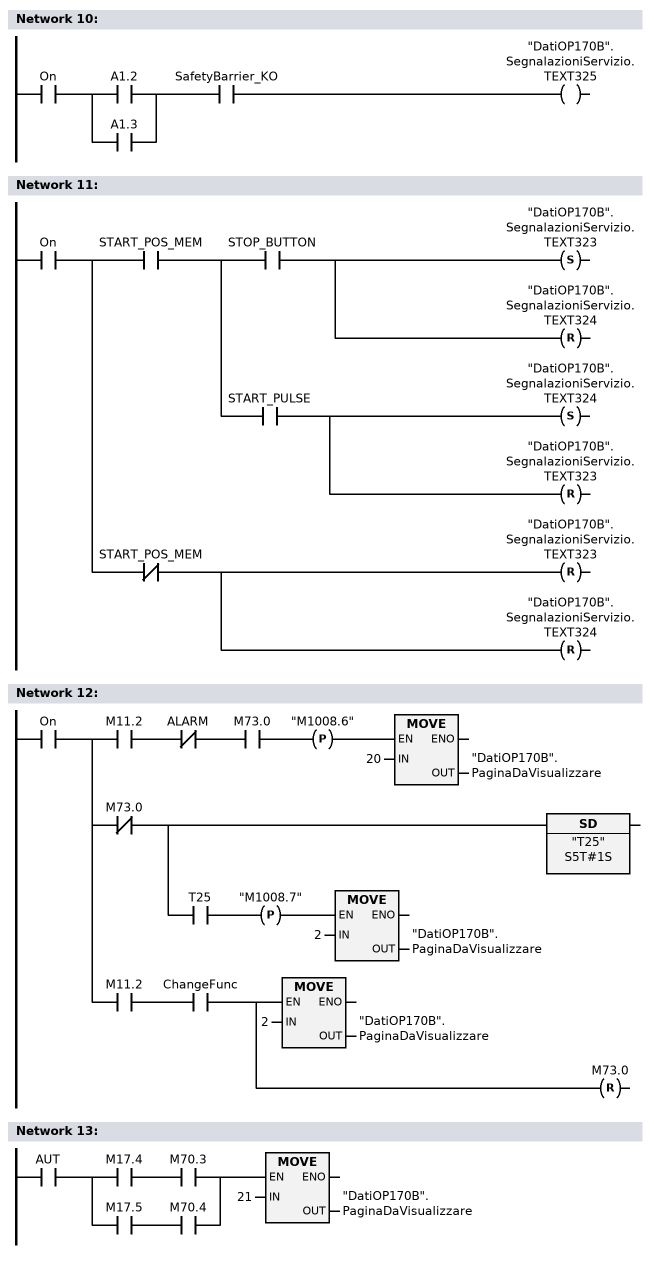
NETWORK
TITLE =
      A     "On";
      A(;
      O     "A1.2";
      O     "A1.3";
      );
      A     "SafetyBarrier_KO";
      =     "DatiOP170B".SegnalazioniServizio.TEXT325;
NETWORK
TITLE =
      A     "On";
      =     L 0.0;
      A     L 0.0;
      A     "START_POS_MEM";
      =     L 0.1;
      A     L 0.1;
      A     "STOP_BUTTON";
      S     "DatiOP170B".SegnalazioniServizio.TEXT323;
      R     "DatiOP170B".SegnalazioniServizio.TEXT324;
      A     L 0.1;
      A     "START_PULSE";
      S     "DatiOP170B".SegnalazioniServizio.TEXT324;
      R     "DatiOP170B".SegnalazioniServizio.TEXT323;
      A     L 0.0;
      AN    "START_POS_MEM";
      R     "DatiOP170B".SegnalazioniServizio.TEXT323;
      R     "DatiOP170B".SegnalazioniServizio.TEXT324;
NETWORK
TITLE =
      A     "On";
      =     L 0.0;
      A     L 0.0;
      A     "M11.2";
      AN    "ALARM";
      A     "M73.0";
      FP    "M1008.6";
      JNB   M008;
      L     20;
      T     "DatiOP170B".PaginaDaVisualizzare;
M008: NOP   0;
      A     L 0.0;
      AN    "M73.0";
      =     L 0.1;
      A     L 0.1;
      BLD   102;
      L     S5T#1S;
      SD    "T25";
      A     L 0.1;
      A     "T25";
      FP    "M1008.7";
      JNB   M009;
      L     2;
      T     "DatiOP170B".PaginaDaVisualizzare;
M009: NOP   0;
      A     L 0.0;
      A     "M11.2";
      A     "ChangeFunc";
      =     L 0.1;
      A     L 0.1;
      JNB   M010;
      L     2;
      T     "DatiOP170B".PaginaDaVisualizzare;
M010: NOP   0;
      A     L 0.1;
      BLD   102;
      R     "M73.0";
NETWORK
TITLE =
      A     "AUT";
      A(;
      A     "M17.4";
      A     "M70.3";
      O;
      A     "M17.5";
      A     "M70.4";
      );
      JNB   M011;
      L     21;
      T     "DatiOP170B".PaginaDaVisualizzare;
M011: NOP   0;
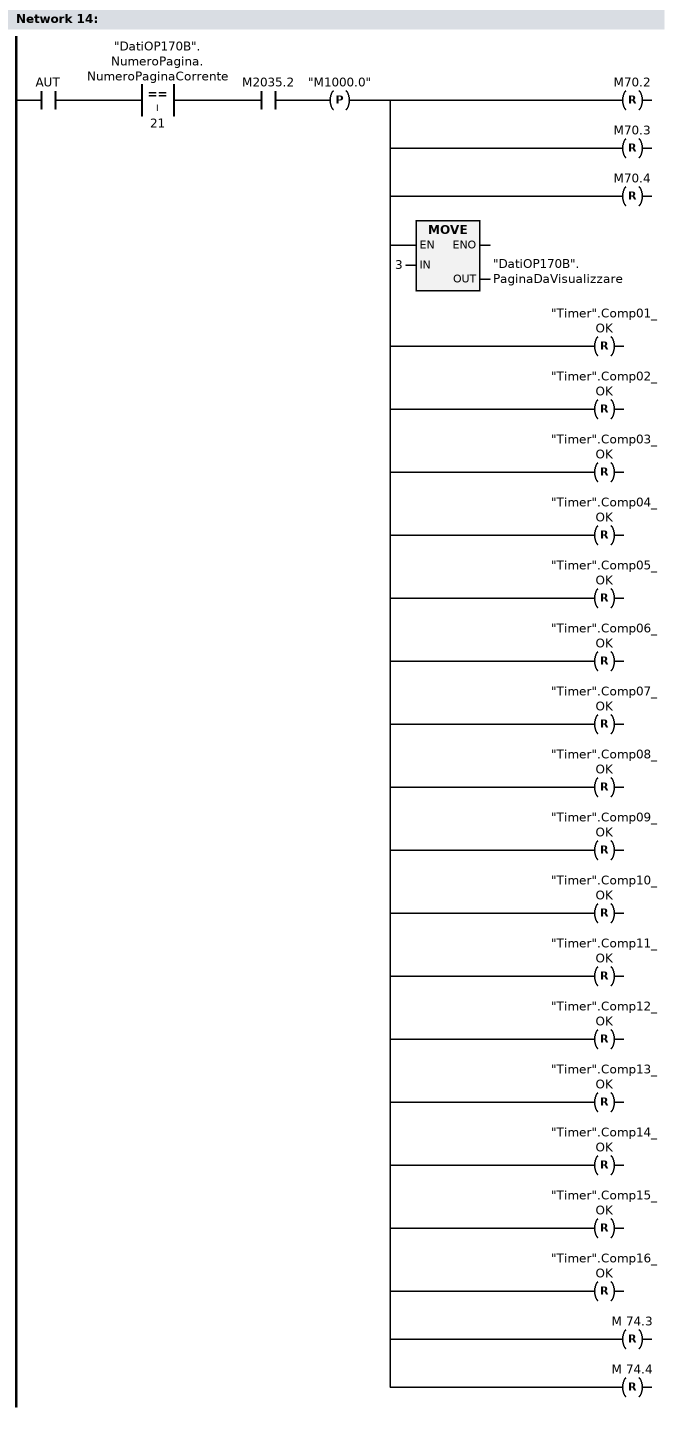
NETWORK
TITLE =
      A     "AUT";
      A(;
      L     "DatiOP170B".NumeroPagina.NumeroPaginaCorrente;
      L     21;
      ==I;
      );
      A     "M2035.2";
      FP    "M1000.0";
      =     L 0.0;
      A     L 0.0;
      BLD   102;
      R     "M70.2";
      A     L 0.0;
      BLD   102;
      R     "M70.3";
      A     L 0.0;
      BLD   102;
      R     "M70.4";
      A     L 0.0;
      JNB   M012;
      L     3;
      T     "DatiOP170B".PaginaDaVisualizzare;
M012: NOP   0;
      A     L 0.0;
      BLD   102;
      R     "Timer".Comp01_OK;
      A     L 0.0;
      BLD   102;
      R     "Timer".Comp02_OK;
      A     L 0.0;
      BLD   102;
      R     "Timer".Comp03_OK;
      A     L 0.0;
      BLD   102;
      R     "Timer".Comp04_OK;
      A     L 0.0;
      BLD   102;
      R     "Timer".Comp05_OK;
      A     L 0.0;
      BLD   102;
      R     "Timer".Comp06_OK;
      A     L 0.0;
      BLD   102;
      R     "Timer".Comp07_OK;
      A     L 0.0;
      BLD   102;
      R     "Timer".Comp08_OK;
      A     L 0.0;
      BLD   102;
      R     "Timer".Comp09_OK;
      A     L 0.0;
      BLD   102;
      R     "Timer".Comp10_OK;
      A     L 0.0;
      BLD   102;
      R     "Timer".Comp11_OK;
      A     L 0.0;
      BLD   102;
      R     "Timer".Comp12_OK;
      A     L 0.0;
      BLD   102;
      R     "Timer".Comp13_OK;
      A     L 0.0;
      BLD   102;
      R     "Timer".Comp14_OK;
      A     L 0.0;
      BLD   102;
      R     "Timer".Comp15_OK;
      A     L 0.0;
      BLD   102;
      R     "Timer".Comp16_OK;
      A     L 0.0;
      BLD   102;
      R     M 74.3;
      A     L 0.0;
      BLD   102;
      R     M 74.4;
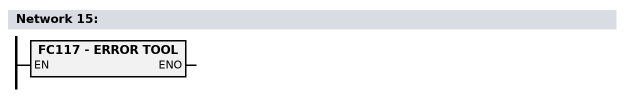
NETWORK
TITLE =
      CALL  "FC117 - ERROR TOOL";
      NOP   0;
END_FUNCTION

FUNCTION "FC18 - OUTPUTS" : VOID	// FC 18
VERSION : 0.1
BEGIN
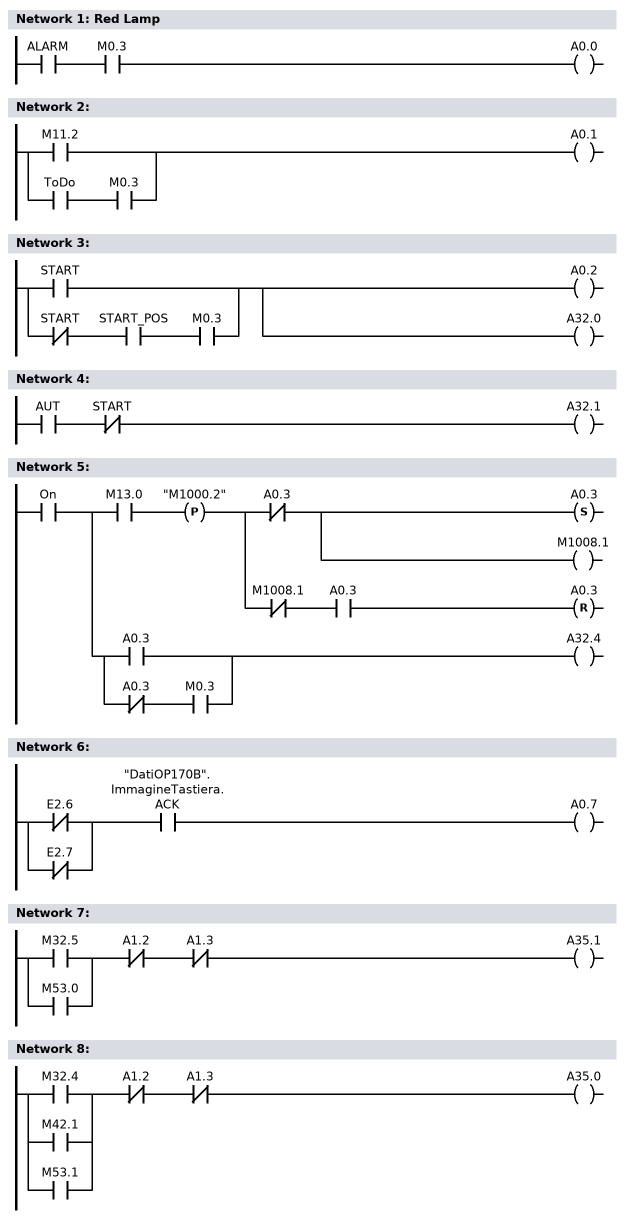
NETWORK
TITLE = Red Lamp
      A     "ALARM";
      A     "M0.3";
      =     "A0.0";
NETWORK
TITLE =
      O     "M11.2";
      O;
      A     "ToDo";
      A     "M0.3";
      =     "A0.1";
NETWORK
TITLE =
      O     "START";
      O;
      AN    "START";
      A     "START_POS";
      A     "M0.3";
      =     "A0.2";
      =     "A32.0";
NETWORK
TITLE =
      A     "AUT";
      AN    "START";
      =     "A32.1";
NETWORK
TITLE =
      A     "On";
      =     L 0.0;
      A     L 0.0;
      A     "M13.0";
      FP    "M1000.2";
      =     L 0.1;
      A     L 0.1;
      AN    "A0.3";
      S     "A0.3";
      =     "M1008.1";
      A     L 0.1;
      AN    "M1008.1";
      A     "A0.3";
      R     "A0.3";
      A     L 0.0;
      A(;
      O     "A0.3";
      O;
      AN    "A0.3";
      A     "M0.3";
      );
      =     "A32.4";
NETWORK
TITLE =
      A(;
      ON    "E2.6";
      ON    "E2.7";
      );
      A     "DatiOP170B".ImmagineTastiera.ACK;
      =     "A0.7";
NETWORK
TITLE =
      A(;
      O     "M32.5";
      O     "M53.0";
      );
      AN    "A1.2";
      AN    "A1.3";
      =     "A35.1";
NETWORK
TITLE =
      A(;
      O     "M32.4";
      O     "M42.1";
      O     "M53.1";
      );
      AN    "A1.2";
      AN    "A1.3";
      =     "A35.0";
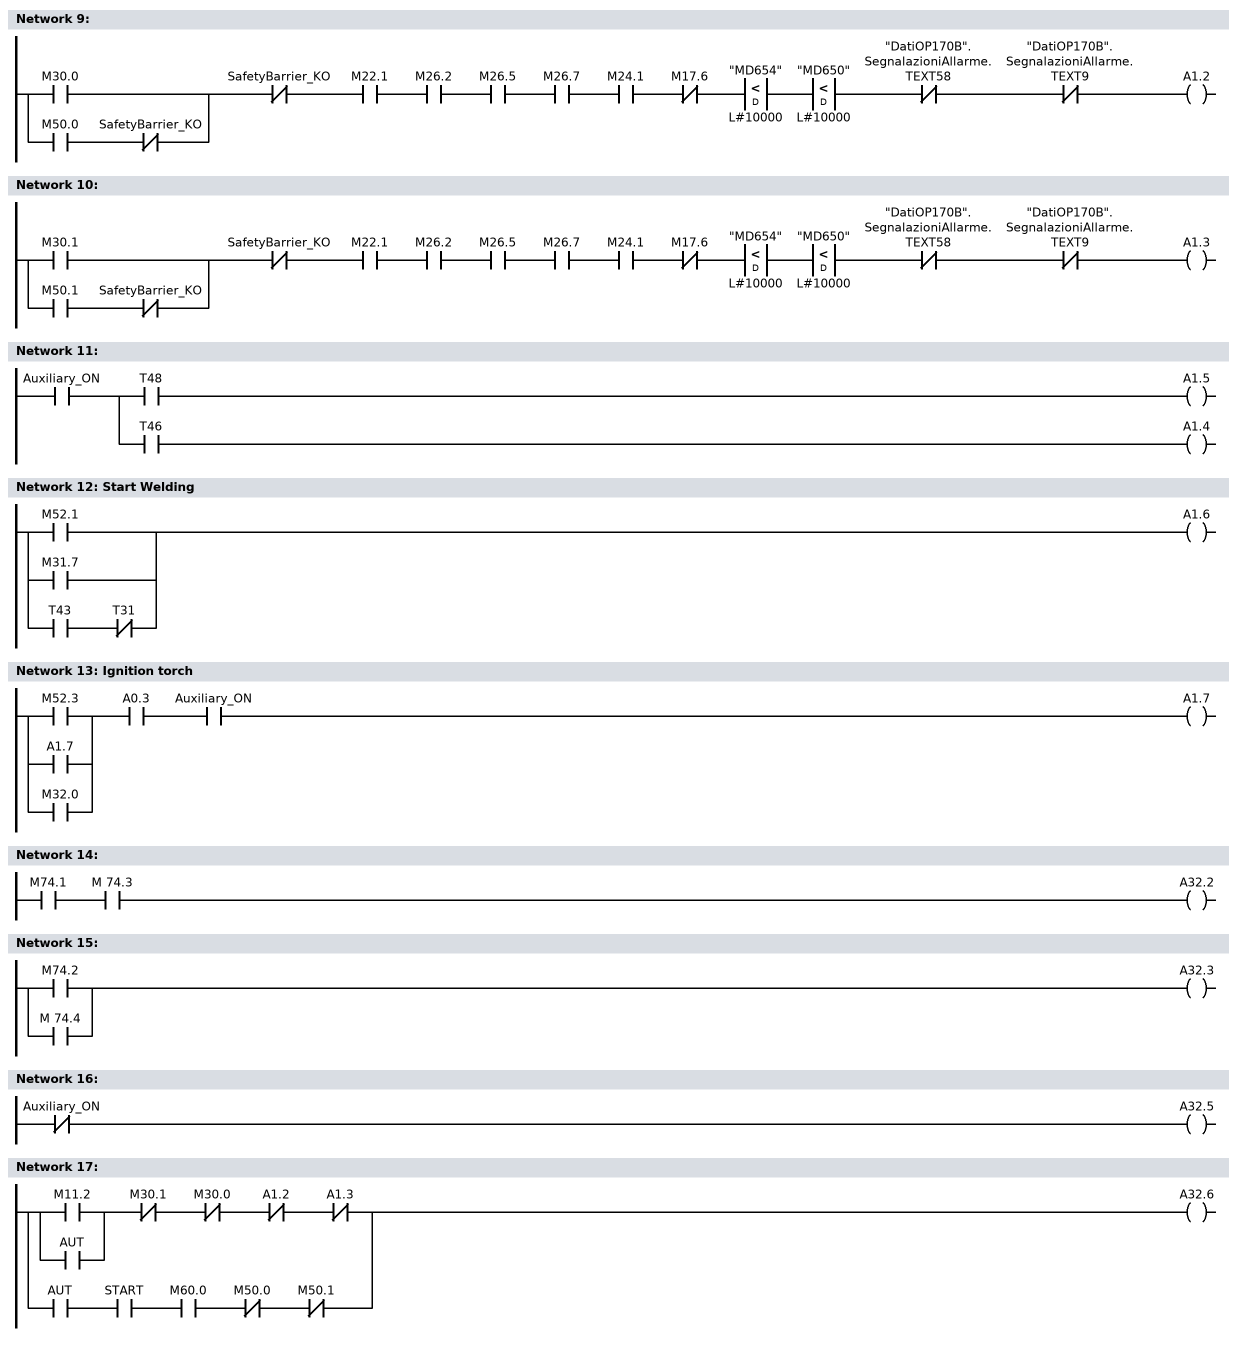
NETWORK
TITLE =
      A(;
      O     "M30.0";
      O;
      A     "M50.0";
      AN    "SafetyBarrier_KO";
      );
      AN    "SafetyBarrier_KO";
      A     "M22.1";
      A     "M26.2";
      A     "M26.5";
      A     "M26.7";
      A     "M24.1";
      AN    "M17.6";
      A(;
      L     "MD654";
      L     L#10000;
      <D;
      );
      A(;
      L     "MD650";
      L     L#10000;
      <D;
      );
      AN    "DatiOP170B".SegnalazioniAllarme.TEXT58;
      AN    "DatiOP170B".SegnalazioniAllarme.TEXT9;
      =     "A1.2";
NETWORK
TITLE =
      A(;
      O     "M30.1";
      O;
      A     "M50.1";
      AN    "SafetyBarrier_KO";
      );
      AN    "SafetyBarrier_KO";
      A     "M22.1";
      A     "M26.2";
      A     "M26.5";
      A     "M26.7";
      A     "M24.1";
      AN    "M17.6";
      A(;
      L     "MD654";
      L     L#10000;
      <D;
      );
      A(;
      L     "MD650";
      L     L#10000;
      <D;
      );
      AN    "DatiOP170B".SegnalazioniAllarme.TEXT58;
      AN    "DatiOP170B".SegnalazioniAllarme.TEXT9;
      =     "A1.3";
NETWORK
TITLE =
      A     "Auxiliary_ON";
      =     L 0.0;
      A     L 0.0;
      A     "T48";
      =     "A1.5";
      A     L 0.0;
      A     "T46";
      =     "A1.4";
NETWORK
TITLE = Start Welding
      O     "M52.1";
      O     "M31.7";
      O;
      A     "T43";
      AN    "T31";
      =     "A1.6";
NETWORK
TITLE = Ignition torch
      A(;
      O     "M52.3";
      O     "A1.7";
      O     "M32.0";
      );
      A     "A0.3";
      A     "Auxiliary_ON";
      =     "A1.7";
NETWORK
TITLE =
      A     "M74.1";
      A     M 74.3;
      =     "A32.2";
NETWORK
TITLE =
      O     "M74.2";
      O     M 74.4;
      =     "A32.3";
NETWORK
TITLE =
      AN    "Auxiliary_ON";
      =     "A32.5";
NETWORK
TITLE =
      A(;
      O     "M11.2";
      O     "AUT";
      );
      AN    "M30.1";
      AN    "M30.0";
      AN    "A1.2";
      AN    "A1.3";
      O;
      A     "AUT";
      A     "START";
      A     "M60.0";
      AN    "M50.0";
      AN    "M50.1";
      =     "A32.6";
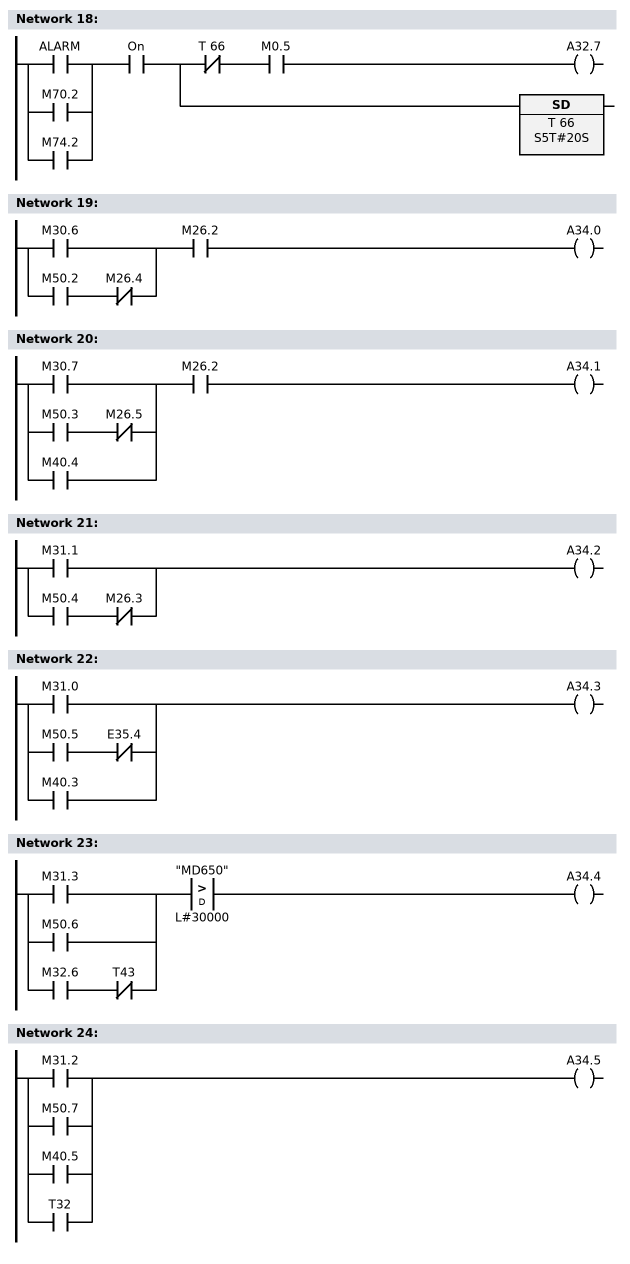
NETWORK
TITLE =
      A(;
      O     "ALARM";
      O     "M70.2";
      O     "M74.2";
      );
      A     "On";
      =     L 0.0;
      A     L 0.0;
      AN    T 66;
      A     "M0.5";
      =     "A32.7";
      A     L 0.0;
      BLD   102;
      L     S5T#20S;
      SD    T 66;
NETWORK
TITLE =
      A(;
      O     "M30.6";
      O;
      A     "M50.2";
      AN    "M26.4";
      );
      A     "M26.2";
      =     "A34.0";
NETWORK
TITLE =
      A(;
      O     "M30.7";
      O;
      A     "M50.3";
      AN    "M26.5";
      O     "M40.4";
      );
      A     "M26.2";
      =     "A34.1";
NETWORK
TITLE =
      O     "M31.1";
      O;
      A     "M50.4";
      AN    "M26.3";
      =     "A34.2";
NETWORK
TITLE =
      O     "M31.0";
      O;
      A     "M50.5";
      AN    "E35.4";
      O     "M40.3";
      =     "A34.3";
NETWORK
TITLE =
      A(;
      O     "M31.3";
      O     "M50.6";
      O;
      A     "M32.6";
      AN    "T43";
      );
      A(;
      L     "MD650";
      L     L#30000;
      >D;
      );
      =     "A34.4";
NETWORK
TITLE =
      O     "M31.2";
      O     "M50.7";
      O     "M40.5";
      O     "T32";
      =     "A34.5";
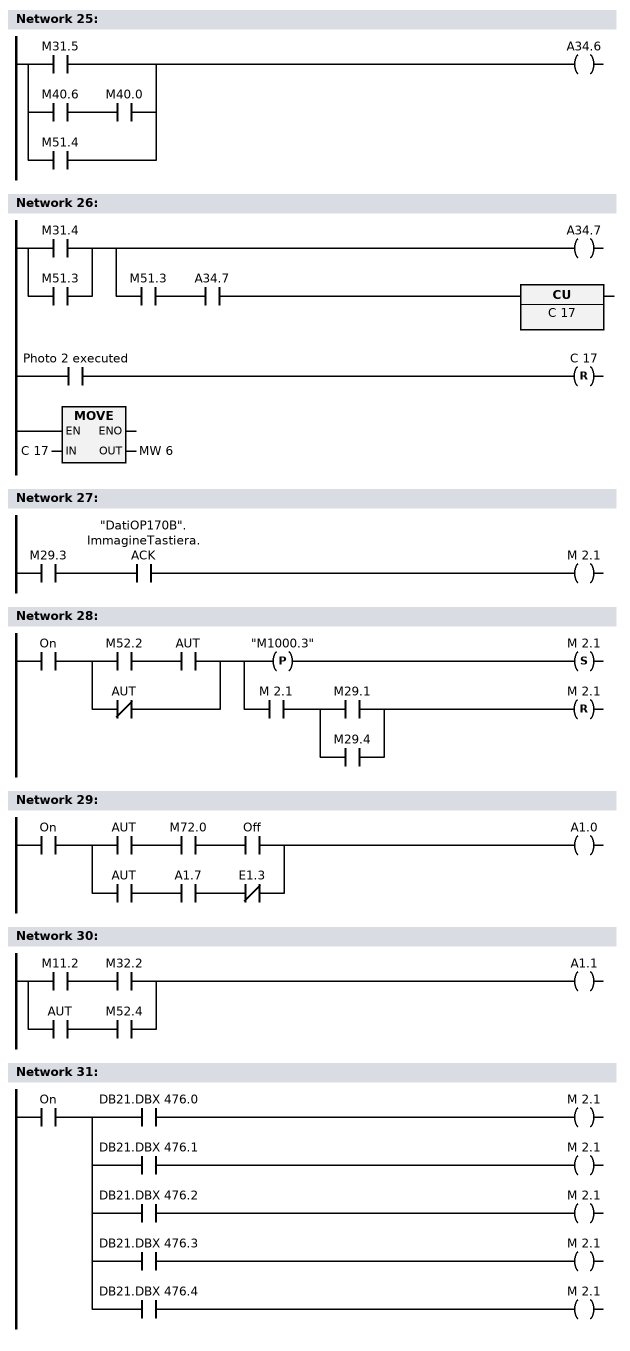
NETWORK
TITLE =
      O     "M31.5";
      O;
      A     "M40.6";
      A     "M40.0";
      O     "M51.4";
      =     "A34.6";
NETWORK
TITLE =
      O     "M31.4";
      O     "M51.3";
      =     L 0.0;
      A     L 0.0;
      BLD   102;
      =     "A34.7";
      A     L 0.0;
      A     "M51.3";
      A     "A34.7";
      CU    C 17;
      BLD   101;
      NOP   0;
      NOP   0;
      A     "Photo 2 executed";
      R     C 17;
      L     C 17;
      T     MW 6;
      NOP   0;
      NOP   0;
NETWORK
TITLE =
      A     "M29.3";
      A     "DatiOP170B".ImmagineTastiera.ACK;
      =     M 2.1;
NETWORK
TITLE =
      A     "On";
      A(;
      A     "M52.2";
      A     "AUT";
      ON    "AUT";
      );
      =     L 0.0;
      A     L 0.0;
      FP    "M1000.3";
      S     M 2.1;
      A     L 0.0;
      A     M 2.1;
      A(;
      O     "M29.1";
      O     "M29.4";
      );
      R     M 2.1;
NETWORK
TITLE =
      A     "On";
      A(;
      A     "AUT";
      A     "M72.0";
      A     "Off";
      O;
      A     "AUT";
      A     "A1.7";
      AN    "E1.3";
      );
      =     "A1.0";
NETWORK
TITLE =
      A     "M11.2";
      A     "M32.2";
      O;
      A     "AUT";
      A     "M52.4";
      =     "A1.1";
NETWORK
TITLE =
      A     "On";
      =     L 0.0;
      A     L 0.0;
      A     DB21.DBX 476.0;
      =     M 2.1;
      A     L 0.0;
      A     DB21.DBX 476.1;
      =     M 2.1;
      A     L 0.0;
      A     DB21.DBX 476.2;
      =     M 2.1;
      A     L 0.0;
      A     DB21.DBX 476.3;
      =     M 2.1;
      A     L 0.0;
      A     DB21.DBX 476.4;
      =     M 2.1;
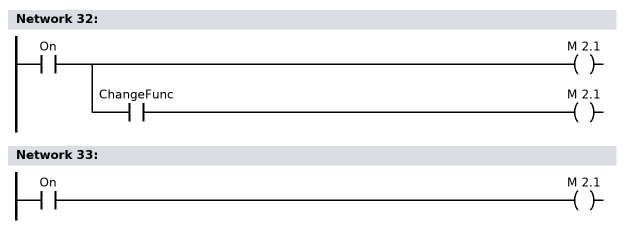
NETWORK
TITLE =
      A     "On";
      =     L 0.0;
      A     L 0.0;
      BLD   102;
      =     M 2.1;
      A     L 0.0;
      A     "ChangeFunc";
      =     M 2.1;
NETWORK
TITLE =
      A     "On";
      =     M 2.1;
END_FUNCTION

FUNCTION "FC19 - REPOSITIONING" : VOID	// FC 19
VERSION : 0.1
BEGIN
// (block stored without names or comments; labels and parameter names are numbered)
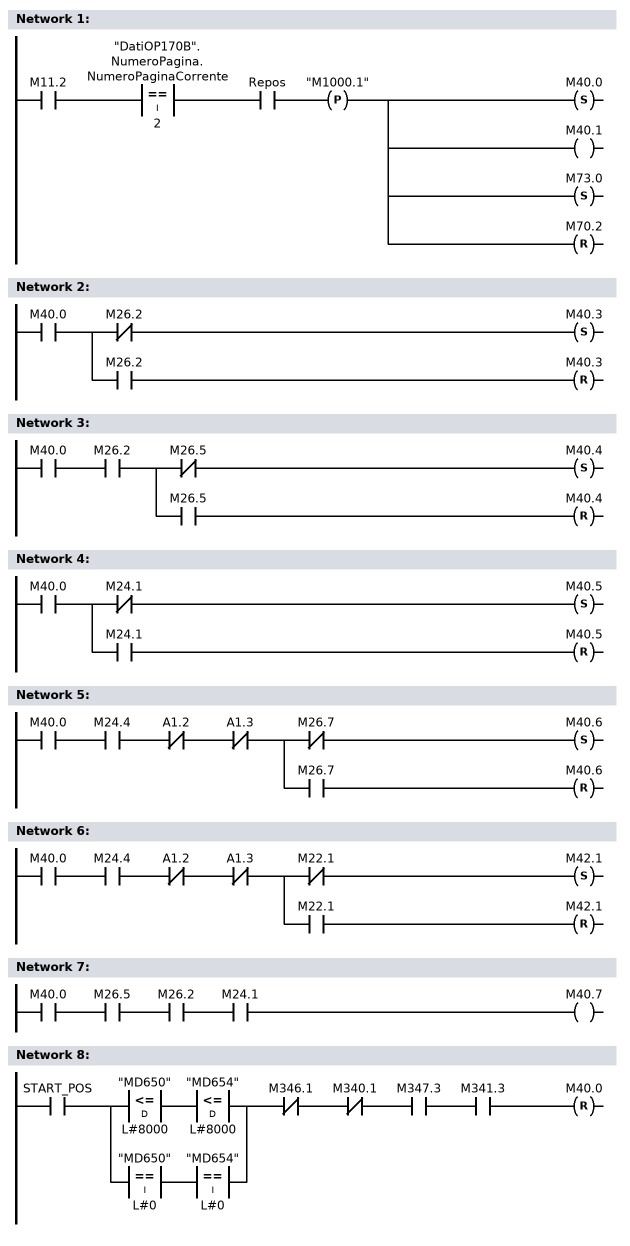
NETWORK
TITLE =
      A     "M11.2";
      A(;
      L     "DatiOP170B".NumeroPagina.NumeroPaginaCorrente;
      L     2;
      ==I;
      );
      A     "Repos";
      FP    "M1000.1";
      S     "M40.0";
      =     "M40.1";
      S     "M73.0";
      R     "M70.2";
NETWORK
TITLE =
      A     "M40.0";
      =     L 0.0;
      A     L 0.0;
      AN    "M26.2";
      S     "M40.3";
      A     L 0.0;
      A     "M26.2";
      R     "M40.3";
NETWORK
TITLE =
      A     "M40.0";
      A     "M26.2";
      =     L 0.0;
      A     L 0.0;
      AN    "M26.5";
      S     "M40.4";
      A     L 0.0;
      A     "M26.5";
      R     "M40.4";
NETWORK
TITLE =
      A     "M40.0";
      =     L 0.0;
      A     L 0.0;
      AN    "M24.1";
      S     "M40.5";
      A     L 0.0;
      A     "M24.1";
      R     "M40.5";
NETWORK
TITLE =
      A     "M40.0";
      A     "M24.4";
      AN    "A1.2";
      AN    "A1.3";
      =     L 0.0;
      A     L 0.0;
      AN    "M26.7";
      S     "M40.6";
      A     L 0.0;
      A     "M26.7";
      R     "M40.6";
NETWORK
TITLE =
      A     "M40.0";
      A     "M24.4";
      AN    "A1.2";
      AN    "A1.3";
      =     L 0.0;
      A     L 0.0;
      AN    "M22.1";
      S     "M42.1";
      A     L 0.0;
      A     "M22.1";
      R     "M42.1";
NETWORK
TITLE =
      A     "M40.0";
      A     "M26.5";
      A     "M26.2";
      A     "M24.1";
      =     "M40.7";
NETWORK
TITLE =
      A     "START_POS";
      A(;
      A(;
      L     "MD650";
      L     L#8000;
      <=D;
      );
      A(;
      L     "MD654";
      L     L#8000;
      <=D;
      );
      O;
      A(;
      L     "MD650";
      L     L#0;
      ==I;
      );
      A(;
      L     "MD654";
      L     L#0;
      ==I;
      );
      );
      AN    "M346.1";
      AN    "M340.1";
      A     "M347.3";
      A     "M341.3";
      R     "M40.0";
NETWORK
TITLE =
END_FUNCTION

FUNCTION "FC - AUTOMATIC" : VOID	// FC 24
VERSION : 0.1
BEGIN
// (block stored without names or comments; labels and parameter names are numbered)
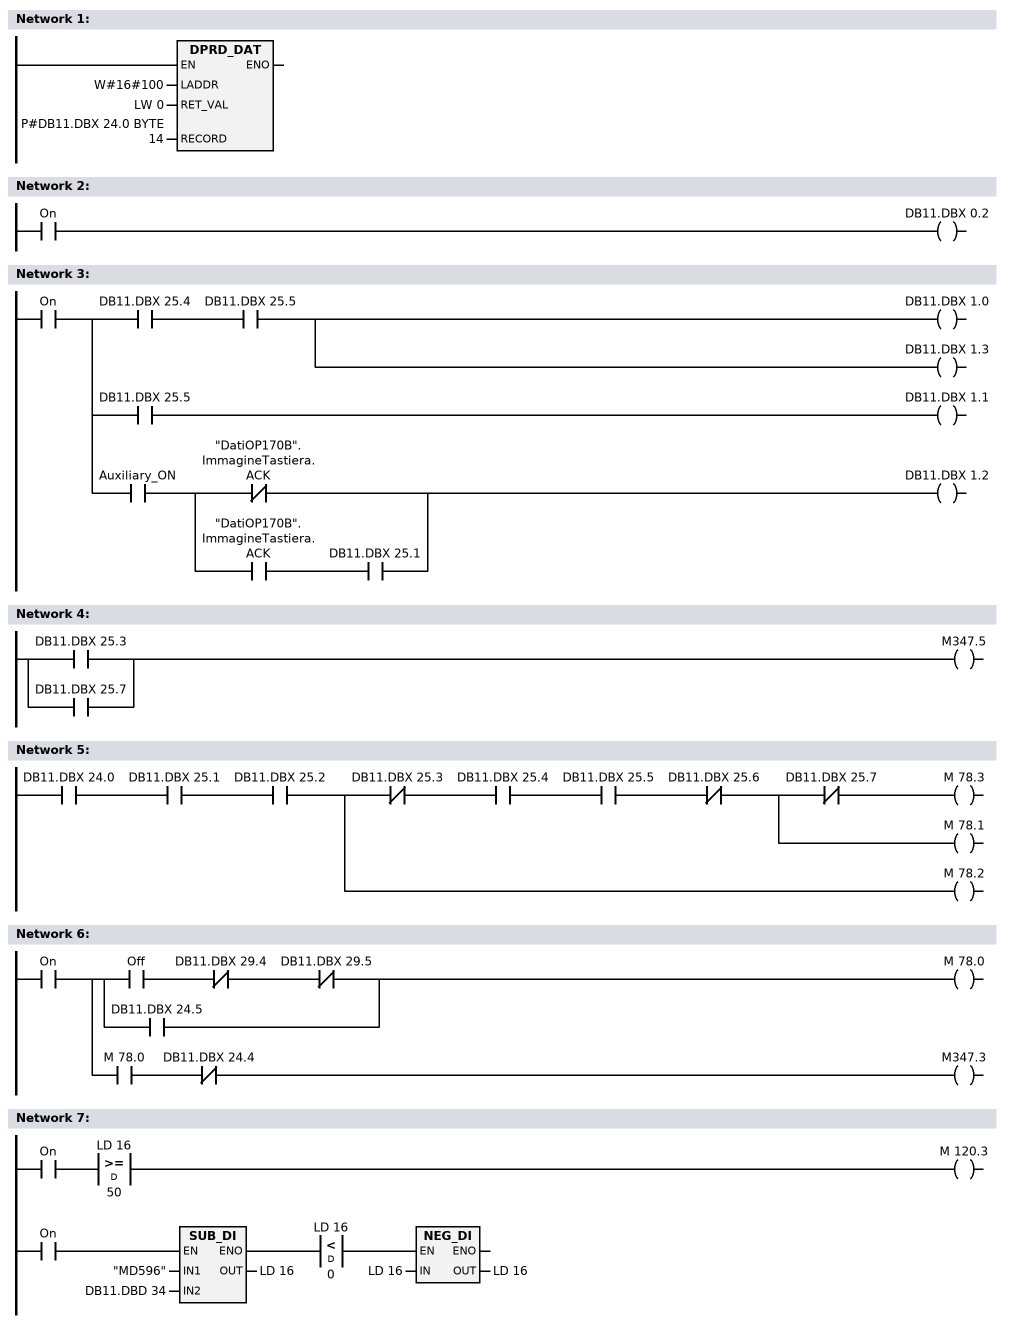
NETWORK
TITLE =
      CALL  "DPRD_DAT" (
           LADDR                    := W#16#100,
           RET_VAL                  := LW 0,
           RECORD                   := P#DB11.DBX 24.0 BYTE 14);
      NOP   0;
NETWORK
TITLE =
      A     "On";
      =     DB11.DBX 0.2;
NETWORK
TITLE =
      A     "On";
      =     L 21.0;
      A     L 21.0;
      A     DB11.DBX 25.4;
      A     DB11.DBX 25.5;
      =     DB11.DBX 1.0;
      =     DB11.DBX 1.3;
      A     L 21.0;
      A     DB11.DBX 25.5;
      =     DB11.DBX 1.1;
      A     L 21.0;
      A     "Auxiliary_ON";
      A(;
      ON    "DatiOP170B".ImmagineTastiera.ACK;
      O;
      A     "DatiOP170B".ImmagineTastiera.ACK;
      A     DB11.DBX 25.1;
      );
      =     DB11.DBX 1.2;
NETWORK
TITLE =
      O     DB11.DBX 25.3;
      O     DB11.DBX 25.7;
      =     "M347.5";
NETWORK
TITLE =
      A     DB11.DBX 24.0;
      A     DB11.DBX 25.1;
      A     DB11.DBX 25.2;
      =     L 21.0;
      A     L 21.0;
      AN    DB11.DBX 25.3;
      A     DB11.DBX 25.4;
      A     DB11.DBX 25.5;
      AN    DB11.DBX 25.6;
      =     L 21.1;
      A     L 21.1;
      AN    DB11.DBX 25.7;
      =     M 78.3;
      A     L 21.1;
      BLD   102;
      =     M 78.1;
      A     L 21.0;
      BLD   102;
      =     M 78.2;
NETWORK
TITLE =
      A     "On";
      =     L 21.0;
      A     L 21.0;
      A(;
      A     "Off";
      AN    DB11.DBX 29.4;
      AN    DB11.DBX 29.5;
      O     DB11.DBX 24.5;
      );
      =     M 78.0;
      A     L 21.0;
      A     M 78.0;
      AN    DB11.DBX 24.4;
      =     "M347.3";
NETWORK
TITLE =
      A     "On";
      =     L 20.0;
      A(;
      A     L 20.0;
      JNB   M001;
      L     "MD596";
      L     DB11.DBD 34;
      -D;
      T     LD 16;
      AN    OV;
      SAVE;
      CLR;
M001: A     BR;
      );
      A(;
      L     LD 16;
      L     0;
      <D;
      );
      JNB   M002;
      L     LD 16;
      NEGD;
      T     LD 16;
M002: NOP   0;
      A     L 20.0;
      A(;
      L     LD 16;
      L     50;
      >=D;
      );
      =     M 120.3;
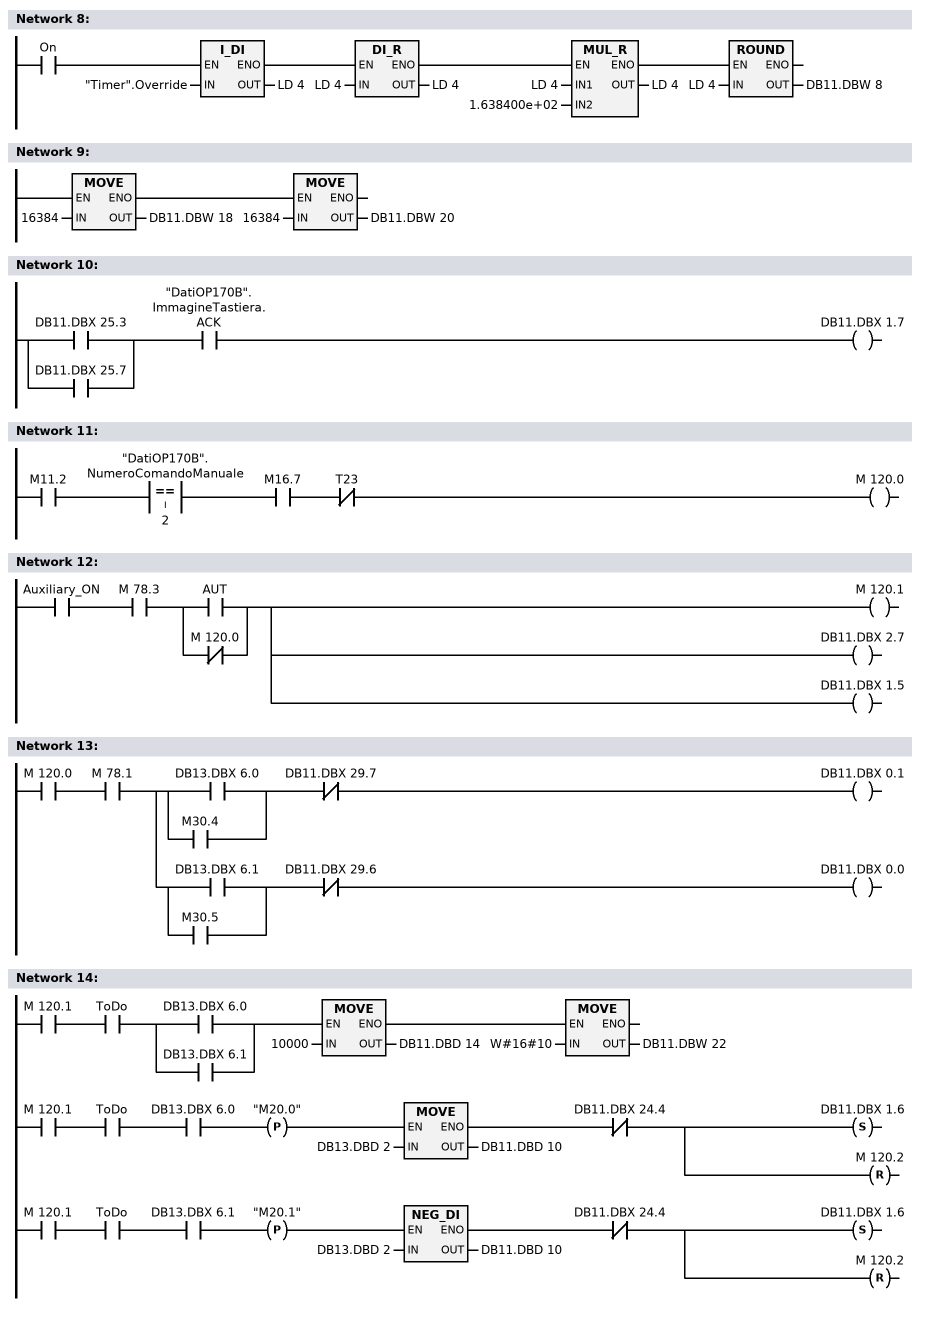
NETWORK
TITLE =
      A(;
      A(;
      A(;
      A     "On";
      JNB   M003;
      L     "Timer".Override;
      ITD;
      T     LD 4;
      SET;
      SAVE;
      CLR;
M003: A     BR;
      );
      JNB   M004;
      L     LD 4;
      DTR;
      T     LD 4;
      SET;
      SAVE;
      CLR;
M004: A     BR;
      );
      JNB   M005;
      L     LD 4;
      L     1.638400e+02;
      *R;
      T     LD 4;
      AN    OV;
      SAVE;
      CLR;
M005: A     BR;
      );
      JNB   M006;
      L     LD 4;
      RND;
      T     DB11.DBW 8;
M006: NOP   0;
NETWORK
TITLE =
      A(;
      L     16384;
      T     DB11.DBW 18;
      SET;
      SAVE;
      CLR;
      A     BR;
      );
      JNB   M007;
      L     16384;
      T     DB11.DBW 20;
M007: NOP   0;
NETWORK
TITLE =
      A(;
      O     DB11.DBX 25.3;
      O     DB11.DBX 25.7;
      );
      A     "DatiOP170B".ImmagineTastiera.ACK;
      =     DB11.DBX 1.7;
NETWORK
TITLE =
      A     "M11.2";
      A(;
      L     "DatiOP170B".NumeroComandoManuale;
      L     2;
      ==I;
      );
      A     "M16.7";
      AN    "T23";
      =     M 120.0;
NETWORK
TITLE =
      A     "Auxiliary_ON";
      A     M 78.3;
      A(;
      O     "AUT";
      ON    M 120.0;
      );
      =     M 120.1;
      =     DB11.DBX 2.7;
      =     DB11.DBX 1.5;
NETWORK
TITLE =
      A     M 120.0;
      A     M 78.1;
      =     L 21.0;
      A     L 21.0;
      A(;
      O     DB13.DBX 6.0;
      O     "M30.4";
      );
      AN    DB11.DBX 29.7;
      =     DB11.DBX 0.1;
      A     L 21.0;
      A(;
      O     DB13.DBX 6.1;
      O     "M30.5";
      );
      AN    DB11.DBX 29.6;
      =     DB11.DBX 0.0;
NETWORK
TITLE =
      A     M 120.1;
      A     "ToDo";
      =     L 21.0;
      A(;
      A     L 21.0;
      A(;
      O     DB13.DBX 6.0;
      O     DB13.DBX 6.1;
      );
      JNB   M008;
      L     10000;
      T     DB11.DBD 14;
      SET;
      SAVE;
      CLR;
M008: A     BR;
      );
      JNB   M009;
      L     W#16#10;
      T     DB11.DBW 22;
M009: NOP   0;
      A(;
      A     L 21.0;
      A     DB13.DBX 6.0;
      FP    "M20.0";
      JNB   M010;
      L     DB13.DBD 2;
      T     DB11.DBD 10;
      SET;
      SAVE;
      CLR;
M010: A     BR;
      );
      AN    DB11.DBX 24.4;
      S     DB11.DBX 1.6;
      R     M 120.2;
      A(;
      A     L 21.0;
      A     DB13.DBX 6.1;
      FP    "M20.1";
      JNB   M011;
      L     DB13.DBD 2;
      NEGD;
      T     DB11.DBD 10;
      AN    OV;
      SAVE;
      CLR;
M011: A     BR;
      );
      AN    DB11.DBX 24.4;
      S     DB11.DBX 1.6;
      R     M 120.2;
